// TwinCAT 3 PLC project MU
// ProgramVersion: 3.1.4026.14
// libraries:
//   Tc2_ControllerToolbox, * (Beckhoff Automation GmbH)
//   Tc2_ModbusRTU, * (Beckhoff Automation GmbH)
//   Tc2_SerialCom, * (Beckhoff Automation GmbH)
//   Tc2_Standard, * (Beckhoff Automation GmbH)
//   Tc2_System, * (Beckhoff Automation GmbH)
//   Tc2_Utilities, * (Beckhoff Automation GmbH)
//   Tc3_Module, * (Beckhoff Automation GmbH)
// project tree:
//   DATA TYPES/ E_ComState.TcDUT, E_MFC_INDEX.TcDUT, E_MFC_MESSAGE.TcDUT (not stored), ST_MfcData.TcDUT (not stored)
//   DATA TYPES/MODUELS/ ST_GAS_CABINET.TcDUT (not stored), ST_MAIN_MODULE.TcDUT, ST_NOTIFICATION.TcDUT, ST_NOTIFICATION_MESSAGE.TcDUT (not stored), ST_REACTOR_CABINET.TcDUT, ST_SEQUENCE.TcDUT, ST_SOL_VALVE.TcDUT (not stored), ST_TEMP_CONTROLLER.TcDUT, ST_THROTTLE_VALVE.TcDUT, ST_UTILITY.TcDUT, ST_ROTATION_MOTOR.TcDUT
//   DATA TYPES/PARTS/ ST_ANALOG_PART.TcDUT, ST_DIGITAL_PART.TcDUT, ST_SEQUENCE_PART.TcDUT
//   DEVICE/LINE HEATER/ FB_LINE_HEATER_MANAGER.TcPOU (not stored), FB_Modbus_Send_FIFO.TcPOU (not stored), FB_TEMP_RAMPING.TcPOU
//   DEVICE/LINE HEATER/FUNCTION/ F_Temp_Write_Set_Point.TcPOU (not stored), F_Temp_Write_Value.TcPOU
//   DEVICE/ ST_LineHeater_Data.TcDUT, ST_Modbus_Send_Frame.TcDUT
//   DUTs/ AnalogController.TcDUT, E_ControlMode.TcDUT (not stored), E_RampGeneratorState.TcDUT (not stored), E_RecipeRun.TcDUT (not stored), E_RecipeRunETMode.TcDUT (not stored), E_TowerLamp.TcDUT (not stored), GeneralIO.TcDUT, MainPRGControl.TcDUT, OperationMode.TcDUT (not stored), outWord.TcDUT (not stored), RampGeneratorInput.TcDUT (not stored)
//   DUTs/DUTs/ENUM/ E_aAnalogInputIO_Index.TcDUT, E_AlarmList.TcDUT, E_AlarmSetValue.TcDUT (not stored), E_InputState.TcDUT, E_Interlock.TcDUT, E_Morning_Index.TcDUT, E_WarningList.TcDUT (not stored)
//   DUTs/DUTs/ F_GetReal_USINT.TcDUT
//   DUTs/Interlock/ Interlock.TcDUT, InterlockEnableThreshold.TcDUT, InterlockSetting.TcDUT, InterlockState.TcDUT, LogicalInterlockSubstate.TcDUT
//   DUTs/IO/ AnalogIO.TcDUT, DigitalIO.TcDUT, IO.TcDUT
//   DUTs/Recipe/ Recipe.TcDUT, RecipeControl.TcDUT, RecipeRunET.TcDUT (not stored), RecipeStep.TcDUT, ScaleFactor.TcDUT
//   FUNCTION/ BOOL_TO_STRING_LHeaterON.TcPOU, CheckRangeSigned.TcPOU (not stored), CheckRangeUnsigned.TcPOU (not stored), FB_TON_Pausable.TcPOU (not stored), F_GetDorPressure.TcPOU, F_State_All_Valve_Vent.TcPOU (not stored), HEXSTR_TO_REAL_LHeaterPV.TcPOU (not stored), F_ReactorIndexToAnalogControllerIndex.TcPOU, Real_To_String_LineHeater.TcPOU, Real_To_String_ThermalBath.TcPOU (not stored), USINT_TO_WORD_Bit.TcPOU (not stored), USINT_TO_WORD_jh.TcPOU, WORD_TO_USINT_Bit.TcPOU (not stored)
//   GVLs/ GVL_INTERFACE_UI.TcGVL, GVL_COMMAND_FROM_UI.TcGVL (not stored), GVL_CONSTANT.TcGVL, GVL_DEVICE_NET_E3508.TcGVL, GVL_DEVICE_NET_IQ_PLUS.TcGVL, GVL_IO.TcGVL, GVL.TcGVL, GVL_IO_GAS_CABINET.TcGVL, GVL_IO_REACTOR_CABINET.TcGVL, GVL_IO_VALVE.TcGVL (not stored), GVL_PERSISTENT.TcGVL (not stored), GVL_SEQUENCE.TcGVL (not stored), GVL_Serial.TcGVL
//   / PlcTask.TcTTO (not stored)
//   POUs/ FB_AnalogDeviceRampControl.TcPOU, FB_ControlRampGenerator.TcPOU (not stored), FB_DeviationCheck.TcPOU (not stored), FB_FaultCheck.TcPOU (not stored), FB_OverLimitCheck.TcPOU, FB_RecipeAnalogControlInputSequencer.TcPOU, F_StopAnalogRamping_ForRecipe.TcPOU, FB_SensorLimitCheck.TcPOU (not stored), FB_ValveControl.TcPOU, F_ResetTimersAndRCPTimes.TcPOU (not stored), MAIN.TcPOU, P11_E3508.TcPOU, P12_IQ_PLUS.TcPOU, P13_LineHeater.TcPOU, P14_ThermalBath.TcPOU, P15_RotationOperation.TcPOU, P16_CoverOperation.TcPOU, P17_DOROperation.TcPOU, P22_Background_ThermalBath.TcPOU, P30_ManualControl.TcPOU (not stored), P31_PriorityControl.TcPOU, P50_RecipeControl.TcPOU, P60_UpdatePV.TcPOU, P70_Interface.TcPOU (not stored), P90_Interlock.TcPOU, P91_Monitoring.TcPOU, P92_Maintenance.TcPOU
//   POUs/FUNCTION/ FB_RINGBUFFER.TcPOU, F_StateValve_Process_Source.TcPOU, F_StateValve_Process.TcPOU
//   POUs/VARIABLE_LINK/ F_Variable_DeviceLink.TcPOU, F_Variable_Valve.TcPOU, F_Variable_FromUI.TcPOU, F_Variable_FromUI_Interlock.TcPOU, F_Variable_TODevice.TcPOU (not stored), F_Variable_ToUI_InputState.TcPOU
// real-time tasks:
//   TASK PlcTask: cycle T#10ms, priority 20, ADS port 350
// I/O:
//   DEVICE Device 1 (EtherCAT) (disabled), AmsNetId 192.168.123.106.2.1
//     Term 1 (EK1200) [EK1200-5000 EtherCAT Power supply (2A E-Bus)]
//       Term 2 (EL1088) [EL1088 8Ch. Dig. Input 24V, 3ms, negative]
//       Term 3 (EL1088) [EL1088 8Ch. Dig. Input 24V, 3ms, negative]
//       Term 4 (EL1088) [EL1088 8Ch. Dig. Input 24V, 3ms, negative]
//       Term 5 (EL1088) [EL1088 8Ch. Dig. Input 24V, 3ms, negative]
//       Term 6 (EL1088) [EL1088 8Ch. Dig. Input 24V, 3ms, negative]
//       Term 7 (EL1088) [EL1088 8Ch. Dig. Input 24V, 3ms, negative]
//       Term 8 (EL2088) [EL2088 8Ch. Dig. Output 24V, 0.5A, switching to negative]
//       Term 9 (EL2088) [EL2088 8Ch. Dig. Output 24V, 0.5A, switching to negative]
//       Term 10 (EL3064) [EL3064 4Ch. Ana. Input 0-10V]
//       Term 11 (EL4004) [EL4004 4Ch. Ana. Output 0-10V, 12bit]
//       Term 12 (EL9410) [EL9410 E-Bus Power Supplier  (Diagnostics)]
//       Term 13 (EL3064) [EL3064 4Ch. Ana. Input 0-10V]
//       Term 14 (EL4004) [EL4004 4Ch. Ana. Output 0-10V, 12bit]
//       Term 15 (EL3064) [EL3064 4Ch. Ana. Input 0-10V]
//       Term 16 (EL4004) [EL4004 4Ch. Ana. Output 0-10V, 12bit]
//       Term 17 (EL3064) [EL3064 4Ch. Ana. Input 0-10V]
//       Term 18 (EL4004) [EL4004 4Ch. Ana. Output 0-10V, 12bit]
//       Term 19 (EL3102) [EL3102 2Ch. Ana. Input +/-10V, Diff.]
//       Term 20 (EL3024) [EL3024 4Ch. Ana. Input 4-20mA DIFF]
//       Term 21 (EL6021) [EL6021 Interface (RS422/485)]
//       Term 22 (EL6021) [EL6021 Interface (RS422/485)]
//       Term 23 (EL6752) [EL6752 DeviceNet Master]
//       Term 24 (EK1110) [EK1110 EtherCAT extension]
//     Term 25 (EK1100) [EK1100 EtherCAT Coupler (2A E-Bus)]
//       Term 26 (EL1088) [EL1088 8Ch. Dig. Input 24V, 3ms, negative]
//       Term 27 (EL1088) [EL1088 8Ch. Dig. Input 24V, 3ms, negative]
//       Term 28 (EL1088) [EL1088 8Ch. Dig. Input 24V, 3ms, negative]
//       Term 29 (EL2088) [EL2088 8Ch. Dig. Output 24V, 0.5A, switching to negative]
//       Term 30 (EL2088) [EL2088 8Ch. Dig. Output 24V, 0.5A, switching to negative]
//       Term 31 (EL2088) [EL2088 8Ch. Dig. Output 24V, 0.5A, switching to negative]
//       Term 32 (EL3064) [EL3064 4Ch. Ana. Input 0-10V]
//       Term 33 (EL3024) [EL3024 4Ch. Ana. Input 4-20mA DIFF]
//       Term 34 (EL4004) [EL4004 4Ch. Ana. Output 0-10V, 12bit]
//       Term 35 (EL3204) [EL3204 4Ch. Ana. Input PT100 (RTD)]
//       Term 36 (EL9011) [EL9011 End Terminal]
//   DEVICE Device 2 (EL6752) (disabled), AmsNetId 192.168.123.106.3.1
//     SolValve // EDS-File: 'OPP6-2D.EDS' DescText: OPP6-2D Vendor: CKD Corporation Device Type: Generic Device Product Name: OPP6-2D Catalog Number:
//     ThrottleValve // EDS-File: 'TBJQPDNG-L041X01 155OUT154.EDS' DescText: Intellisys IQ-Plus Vendor: Nor-Cal Products Device Type: Process Control Valve Product Name: INTELLISYS Catalog Number: IQ-Plus
//     TempController // EDS-File: '3500-2.3V2.EDS' DescText: Eurotherm 3500 Vendor: Eurotherm Device Type: Generic Product Name: Eurotherm 3500 Catalog Number:
// variable links:
//   MU/MU Instance <-> Device 1 (EtherCAT)/Term 1 (EK1200)/Term 10 (EL3064)
//     PlcTask Inputs/GVL_IO_GAS_CABINET.AI_09_M01_ChalcogenRunPV <-> AI Standard Channel 1/Value
//     PlcTask Inputs/GVL_IO_GAS_CABINET.AI_09_M02_MORunPV <-> AI Standard Channel 2/Value
//     PlcTask Inputs/GVL_IO_GAS_CABINET.AI_09_M03_H2SeSupplyPV <-> AI Standard Channel 3/Value
//     PlcTask Inputs/GVL_IO_GAS_CABINET.AI_09_M04_H2SSupplyPV <-> AI Standard Channel 4/Value
//   MU/MU Instance <-> Device 1 (EtherCAT)/Term 1 (EK1200)/Term 11 (EL4004)
//     PlcTask Outputs/GVL_IO_GAS_CABINET.AO_10_M01_ChalcogenRunSV <-> AO Outputs Channel 1/Analog output
//     PlcTask Outputs/GVL_IO_GAS_CABINET.AO_10_M02_MORunSV <-> AO Outputs Channel 2/Analog output
//     PlcTask Outputs/GVL_IO_GAS_CABINET.AO_10_M03_H2SeSupplySV <-> AO Outputs Channel 3/Analog output
//     PlcTask Outputs/GVL_IO_GAS_CABINET.AO_10_M04_H2SSupplySV <-> AO Outputs Channel 4/Analog output
//   MU/MU Instance <-> Device 1 (EtherCAT)/Term 1 (EK1200)/Term 13 (EL3064)
//     PlcTask Inputs/GVL_IO_GAS_CABINET.AI_11_M05_Source_1TMInSupplyPV <-> AI Standard Channel 1/Value
//     PlcTask Inputs/GVL_IO_GAS_CABINET.AI_11_M06_Source_2TMGaSupplyPV <-> AI Standard Channel 2/Value
//     PlcTask Inputs/GVL_IO_GAS_CABINET.AI_11_M07_Source_3DMSeSupplyPV <-> AI Standard Channel 3/Value
//     PlcTask Inputs/GVL_IO_GAS_CABINET.AI_11_M08_Source_4ChalcoSupplyPV <-> AI Standard Channel 4/Value
//   MU/MU Instance <-> Device 1 (EtherCAT)/Term 1 (EK1200)/Term 14 (EL4004)
//     PlcTask Outputs/GVL_IO_GAS_CABINET.AO_12_M05_Source_1TMInSupplySV <-> AO Outputs Channel 1/Analog output
//     PlcTask Outputs/GVL_IO_GAS_CABINET.AO_12_M06_Source_2TMGaSupplySV <-> AO Outputs Channel 2/Analog output
//     PlcTask Outputs/GVL_IO_GAS_CABINET.AO_12_M07_Source_3DMSeSupplySV <-> AO Outputs Channel 3/Analog output
//     PlcTask Outputs/GVL_IO_GAS_CABINET.AO_12_M08_Source_4ChalcoSupplySV <-> AO Outputs Channel 4/Analog output
//   MU/MU Instance <-> Device 1 (EtherCAT)/Term 1 (EK1200)/Term 15 (EL3064)
//     PlcTask Inputs/GVL_IO_GAS_CABINET.AI_13_M09_LinerPurgePV <-> AI Standard Channel 1/Value
//     PlcTask Inputs/GVL_IO_GAS_CABINET.AI_13_M10_HeaterPurgePV <-> AI Standard Channel 2/Value
//     PlcTask Inputs/GVL_IO_GAS_CABINET.AI_13_M11_ChalcogenVentPV <-> AI Standard Channel 3/Value
//     PlcTask Inputs/GVL_IO_GAS_CABINET.AI_13_M12_MOVentPV <-> AI Standard Channel 4/Value
//   MU/MU Instance <-> Device 1 (EtherCAT)/Term 1 (EK1200)/Term 16 (EL4004)
//     PlcTask Outputs/GVL_IO_GAS_CABINET.AO_14_M09_LinerPurgeSV <-> AO Outputs Channel 1/Analog output
//     PlcTask Outputs/GVL_IO_GAS_CABINET.AO_14_M10_HeaterPurgeSV <-> AO Outputs Channel 2/Analog output
//     PlcTask Outputs/GVL_IO_GAS_CABINET.AO_14_M11_ChalcogenVentSV <-> AO Outputs Channel 3/Analog output
//     PlcTask Outputs/GVL_IO_GAS_CABINET.AO_14_M12_MOVentSV <-> AO Outputs Channel 4/Analog output
//   MU/MU Instance <-> Device 1 (EtherCAT)/Term 1 (EK1200)/Term 17 (EL3064)
//     PlcTask Inputs/GVL_IO_GAS_CABINET.AI_15_E01Source_1TMInPressurePV <-> AI Standard Channel 1/Value
//     PlcTask Inputs/GVL_IO_GAS_CABINET.AI_15_E02Source_2TMGaPressurePV <-> AI Standard Channel 2/Value
//     PlcTask Inputs/GVL_IO_GAS_CABINET.AI_15_E03Source_3DMSePressurePV <-> AI Standard Channel 3/Value
//     PlcTask Inputs/GVL_IO_GAS_CABINET.AI_15_E04Source_4ChalcoPressurePV <-> AI Standard Channel 4/Value
//   MU/MU Instance <-> Device 1 (EtherCAT)/Term 1 (EK1200)/Term 18 (EL4004)
//     PlcTask Outputs/GVL_IO_GAS_CABINET.AO_16_E01Source_1TMInPressureSV <-> AO Outputs Channel 1/Analog output
//     PlcTask Outputs/GVL_IO_GAS_CABINET.AO_16_E02Source_2TMGaPressureSV <-> AO Outputs Channel 2/Analog output
//     PlcTask Outputs/GVL_IO_GAS_CABINET.AO_16_E03Source_3DMSePressureSV <-> AO Outputs Channel 3/Analog output
//     PlcTask Outputs/GVL_IO_GAS_CABINET.AO_16_E04Source_4ChalcoPressureSV <-> AO Outputs Channel 4/Analog output
//   MU/MU Instance <-> Device 1 (EtherCAT)/Term 1 (EK1200)/Term 19 (EL3102)
//     PlcTask Inputs/GVL_IO_GAS_CABINET.DI_17_DP1ChalcogenDP <-> AI Standard Channel 1/Value
//     PlcTask Inputs/GVL_IO_GAS_CABINET.DI_17_DP2MODP <-> AI Standard Channel 2/Value
//   MU/MU Instance <-> Device 1 (EtherCAT)/Term 1 (EK1200)/Term 2 (EL1088)
//     PlcTask Inputs/GVL_IO_GAS_CABINET.DI_01_ControlCabinetDoorClose <-> Channel 5/Input
//     PlcTask Inputs/GVL_IO_GAS_CABINET.DI_01_GasCabinetDoorClose <-> Channel 4/Input
//     PlcTask Inputs/GVL_IO_GAS_CABINET.DI_01_GasCabinetLampButton <-> Channel 2/Input
//     PlcTask Inputs/GVL_IO_GAS_CABINET.DI_01_PneumaticPressureSensor <-> Channel 3/Input
//     PlcTask Inputs/GVL_IO_GAS_CABINET.DI_01_ResetButton <-> Channel 1/Input
//     PlcTask Inputs/GVL_IO_GAS_CABINET.DI_01_SMPS_1Alarm <-> Channel 6/Input
//     PlcTask Inputs/GVL_IO_GAS_CABINET.DI_01_SMPS_2Alarm <-> Channel 7/Input
//     PlcTask Inputs/GVL_IO_GAS_CABINET.DI_01_SMPS_3Alarm <-> Channel 8/Input
//   MU/MU Instance <-> Device 1 (EtherCAT)/Term 1 (EK1200)/Term 20 (EL3024)
//     PlcTask Inputs/GVL_IO_GAS_CABINET.DI_18_S01N2SupplyPressPV <-> AI Standard Channel 1/Value
//     PlcTask Inputs/GVL_IO_GAS_CABINET.DI_18_S02H2SupplyPressPV <-> AI Standard Channel 2/Value
//     PlcTask Inputs/GVL_IO_GAS_CABINET.DI_18_S03H2SSupplyPressPV <-> AI Standard Channel 3/Value
//     PlcTask Inputs/GVL_IO_GAS_CABINET.DI_18_S04H2SeSupplyPressPV <-> AI Standard Channel 4/Value
//   MU/MU Instance <-> Device 1 (EtherCAT)/Term 1 (EK1200)/Term 21 (EL6021)
//     PlcTask Inputs/GVL.fbLineHeater_Manager.fbModbus_Master.InData/D <-> COM TxPDO-Map Inputs/Data In 0
//     PlcTask Inputs/GVL.fbLineHeater_Manager.fbModbus_Master.InData/D @bit {8..168 step 8} <-> COM TxPDO-Map Inputs/Data In {1..21}  (21 links)
//     PlcTask Inputs/GVL.fbLineHeater_Manager.fbModbus_Master.InData/Status <-> COM TxPDO-Map Inputs/Status
//     PlcTask Outputs/GVL.fbLineHeater_Manager.fbModbus_Master.OutData/Ctrl <-> COM RxPDO-Map Outputs/Ctrl
//     PlcTask Outputs/GVL.fbLineHeater_Manager.fbModbus_Master.OutData/D <-> COM RxPDO-Map Outputs/Data Out 0
//     PlcTask Outputs/GVL.fbLineHeater_Manager.fbModbus_Master.OutData/D @bit {8..168 step 8} <-> COM RxPDO-Map Outputs/Data Out {1..21}  (21 links)
//   MU/MU Instance <-> Device 1 (EtherCAT)/Term 1 (EK1200)/Term 22 (EL6021)
//     PlcTask Inputs/GVL_Serial.stIn_KL6031_TB/D <-> COM TxPDO-Map Inputs/Data In 0
//     PlcTask Inputs/GVL_Serial.stIn_KL6031_TB/D @bit {8..168 step 8} <-> COM TxPDO-Map Inputs/Data In {1..21}  (21 links)
//     PlcTask Inputs/GVL_Serial.stIn_KL6031_TB/Status <-> COM TxPDO-Map Inputs/Status
//     PlcTask Outputs/GVL_Serial.stOut_KL6031_TB/Ctrl <-> COM RxPDO-Map Outputs/Ctrl
//     PlcTask Outputs/GVL_Serial.stOut_KL6031_TB/D <-> COM RxPDO-Map Outputs/Data Out 0
//     PlcTask Outputs/GVL_Serial.stOut_KL6031_TB/D @bit {8..168 step 8} <-> COM RxPDO-Map Outputs/Data Out {1..21}  (21 links)
//   MU/MU Instance <-> Device 1 (EtherCAT)/Term 1 (EK1200)/Term 3 (EL1088)
//     PlcTask Inputs/GVL_IO_GAS_CABINET.DI_02_CoverLiftMotorCP <-> Channel 7/Input
//     PlcTask Inputs/GVL_IO_GAS_CABINET.DI_02_GraphiteHeaterELCB <-> Channel 2/Input
//     PlcTask Inputs/GVL_IO_GAS_CABINET.DI_02_LineHeatersELCB <-> Channel 5/Input
//     PlcTask Inputs/GVL_IO_GAS_CABINET.DI_02_RotationMotorCP <-> Channel 6/Input
//     PlcTask Inputs/GVL_IO_GAS_CABINET.DI_02_SMPS_4Alarm <-> Channel 1/Input
//     PlcTask Inputs/GVL_IO_GAS_CABINET.DI_02_T_VCP <-> Channel 8/Input
//     PlcTask Inputs/GVL_IO_GAS_CABINET.DI_02_ThermalBathsELCB <-> Channel 3/Input
//     PlcTask Inputs/GVL_IO_GAS_CABINET.DI_02_VacuumPumpELCB <-> Channel 4/Input
//   MU/MU Instance <-> Device 1 (EtherCAT)/Term 1 (EK1200)/Term 4 (EL1088)
//     PlcTask Inputs/GVL_IO_GAS_CABINET.DI_03_CabinetLampsCP <-> Channel 2/Input
//     PlcTask Inputs/GVL_IO_GAS_CABINET.DI_03_GasDetectorCP <-> Channel 1/Input
//     PlcTask Inputs/GVL_IO_GAS_CABINET.DI_03_LineHeater_1CP <-> Channel 4/Input
//     PlcTask Inputs/GVL_IO_GAS_CABINET.DI_03_LineHeater_2CP <-> Channel 5/Input
//     PlcTask Inputs/GVL_IO_GAS_CABINET.DI_03_LineHeater_3CP <-> Channel 6/Input
//     PlcTask Inputs/GVL_IO_GAS_CABINET.DI_03_LineHeater_4CP <-> Channel 7/Input
//     PlcTask Inputs/GVL_IO_GAS_CABINET.DI_03_LineHeater_5CP <-> Channel 8/Input
//     PlcTask Inputs/GVL_IO_GAS_CABINET.DI_03_MFCPowerCP <-> Channel 3/Input
//   MU/MU Instance <-> Device 1 (EtherCAT)/Term 1 (EK1200)/Term 5 (EL1088)
//     PlcTask Inputs/GVL_IO_GAS_CABINET.DI_04_ExternalScrubberFault <-> Channel 8/Input
//     PlcTask Inputs/GVL_IO_GAS_CABINET.DI_04_FireSensor <-> Channel 7/Input
//     PlcTask Inputs/GVL_IO_GAS_CABINET.DI_04_GasDetectorH2 <-> Channel 4/Input
//     PlcTask Inputs/GVL_IO_GAS_CABINET.DI_04_GasDetectorH2S <-> Channel 5/Input
//     PlcTask Inputs/GVL_IO_GAS_CABINET.DI_04_GasDetectorH2Se <-> Channel 6/Input
//     PlcTask Inputs/GVL_IO_GAS_CABINET.DI_04_LineHeater_6CP <-> Channel 1/Input
//     PlcTask Inputs/GVL_IO_GAS_CABINET.DI_04_LineHeater_7CP <-> Channel 2/Input
//     PlcTask Inputs/GVL_IO_GAS_CABINET.DI_04_LineHeater_8CP <-> Channel 3/Input
//   MU/MU Instance <-> Device 1 (EtherCAT)/Term 1 (EK1200)/Term 6 (EL1088)
//     PlcTask Inputs/GVL_IO_GAS_CABINET.DI_05_ExternalH2GasCabinetFault <-> Channel 1/Input
//     PlcTask Inputs/GVL_IO_GAS_CABINET.DI_05_ExternalH2SGasCabinetFault <-> Channel 2/Input
//     PlcTask Inputs/GVL_IO_GAS_CABINET.DI_05_ExternalH2SeGasCabinetFault <-> Channel 3/Input
//     PlcTask Inputs/GVL_IO_GAS_CABINET.DI_05_ExternalUserInputAlarm <-> Channel 4/Input
//     PlcTask Inputs/GVL_IO_GAS_CABINET.DI_05_ThermalBath_1CutOffAlarm <-> Channel 6/Input
//     PlcTask Inputs/GVL_IO_GAS_CABINET.DI_05_ThermalBath_2CutOffAlarm <-> Channel 8/Input
//     PlcTask Inputs/GVL_IO_GAS_CABINET.DI_05_ThermalBath_1DeviationAlarm <-> Channel 5/Input
//     PlcTask Inputs/GVL_IO_GAS_CABINET.DI_05_ThermalBath_2DeviationAlarm <-> Channel 7/Input
//   MU/MU Instance <-> Device 1 (EtherCAT)/Term 1 (EK1200)/Term 7 (EL1088)
//     PlcTask Inputs/GVL_IO_GAS_CABINET.DI_06_Spare_01 <-> Channel 5/Input
//     PlcTask Inputs/GVL_IO_GAS_CABINET.DI_06_Spare_02 <-> Channel 6/Input
//     PlcTask Inputs/GVL_IO_GAS_CABINET.DI_06_Spare_03 <-> Channel 7/Input
//     PlcTask Inputs/GVL_IO_GAS_CABINET.DI_06_Spare_04 <-> Channel 8/Input
//     PlcTask Inputs/GVL_IO_GAS_CABINET.DI_06_ThermalBath_3CutOffAlarm <-> Channel 2/Input
//     PlcTask Inputs/GVL_IO_GAS_CABINET.DI_06_ThermalBath_4CutOffAlarm <-> Channel 4/Input
//     PlcTask Inputs/GVL_IO_GAS_CABINET.DI_06_ThermalBath_3DeviationAlarm <-> Channel 1/Input
//     PlcTask Inputs/GVL_IO_GAS_CABINET.DI_06_ThermalBath_4DeviationAlarm <-> Channel 3/Input
//   MU/MU Instance <-> Device 1 (EtherCAT)/Term 1 (EK1200)/Term 8 (EL2088)
//     PlcTask Outputs/GVL_IO_GAS_CABINET.DO_07_ControlCabinetLamp <-> Channel 2/Output
//     PlcTask Outputs/GVL_IO_GAS_CABINET.DO_07_GasCabinetLamp <-> Channel 3/Output
//     PlcTask Outputs/GVL_IO_GAS_CABINET.DO_07_GraphiteHeaterMC <-> Channel 4/Output
//     PlcTask Outputs/GVL_IO_GAS_CABINET.DO_07_LineHeatersMC <-> Channel 7/Output
//     PlcTask Outputs/GVL_IO_GAS_CABINET.DO_07_ResetButtonLamp <-> Channel 8/Output
//     PlcTask Outputs/GVL_IO_GAS_CABINET.DO_07_SystemPowerOffLock <-> Channel 1/Output
//     PlcTask Outputs/GVL_IO_GAS_CABINET.DO_07_ThermalBathsMC <-> Channel 5/Output
//     PlcTask Outputs/GVL_IO_GAS_CABINET.DO_07_VacuumPumpMC <-> Channel 6/Output
//   MU/MU Instance <-> Device 1 (EtherCAT)/Term 1 (EK1200)/Term 9 (EL2088)
//     PlcTask Outputs/GVL_IO_GAS_CABINET.DO_08_Spare_01 <-> Channel 1/Output
//     PlcTask Outputs/GVL_IO_GAS_CABINET.DO_08_Spare_02 <-> Channel 2/Output
//     PlcTask Outputs/GVL_IO_GAS_CABINET.DO_08_Spare_03 <-> Channel 3/Output
//     PlcTask Outputs/GVL_IO_GAS_CABINET.DO_08_Spare_04 <-> Channel 4/Output
//     PlcTask Outputs/GVL_IO_GAS_CABINET.DO_08_Spare_05 <-> Channel 5/Output
//     PlcTask Outputs/GVL_IO_GAS_CABINET.DO_08_Spare_06 <-> Channel 6/Output
//     PlcTask Outputs/GVL_IO_GAS_CABINET.DO_08_Spare_07 <-> Channel 7/Output
//     PlcTask Outputs/GVL_IO_GAS_CABINET.DO_08_Spare_08 <-> Channel 8/Output
//   MU/MU Instance <-> Device 1 (EtherCAT)/Term 25 (EK1100)/Term 26 (EL1088)
//     PlcTask Inputs/GVL_IO_REACTOR_CABINET.DI_01_ClampLock <-> Channel 7/Input
//     PlcTask Inputs/GVL_IO_REACTOR_CABINET.DI_01_ClampRelease <-> Channel 8/Input
//     PlcTask Inputs/GVL_IO_REACTOR_CABINET.DI_01_DORATMButton <-> Channel 4/Input
//     PlcTask Inputs/GVL_IO_REACTOR_CABINET.DI_01_DORVACButton <-> Channel 3/Input
//     PlcTask Inputs/GVL_IO_REACTOR_CABINET.DI_01_MaintenanceModeKey <-> Channel 1/Input
//     PlcTask Inputs/GVL_IO_REACTOR_CABINET.DI_01_ReactorCabinetLampButton <-> Channel 2/Input
//     PlcTask Inputs/GVL_IO_REACTOR_CABINET.DI_01_ReactorDoorDownButton <-> Channel 6/Input
//     PlcTask Inputs/GVL_IO_REACTOR_CABINET.DI_01_ReactorDoorUpButton <-> Channel 5/Input
//   MU/MU Instance <-> Device 1 (EtherCAT)/Term 25 (EK1100)/Term 27 (EL1088)
//     PlcTask Inputs/GVL_IO_REACTOR_CABINET.DI_02_C_WFlowSensor <-> Channel 1/Input
//     PlcTask Inputs/GVL_IO_REACTOR_CABINET.DI_02_ReactorDoorUpLimitSensor <-> Channel 8/Input
//     PlcTask Inputs/GVL_IO_REACTOR_CABINET.DI_02_SusceptorRotationMotorFault <-> Channel 2/Input
//     PlcTask Inputs/GVL_IO_REACTOR_CABINET.DI_02_VacuumPumpAlarm <-> Channel 5/Input
//     PlcTask Inputs/GVL_IO_REACTOR_CABINET.DI_02_VacuumPumpFBRunning <-> Channel 7/Input
//     PlcTask Inputs/GVL_IO_REACTOR_CABINET.DI_02_VacuumPumpFail <-> Channel 3/Input
//     PlcTask Inputs/GVL_IO_REACTOR_CABINET.DI_02_VacuumPumpRunning <-> Channel 6/Input
//     PlcTask Inputs/GVL_IO_REACTOR_CABINET.DI_02_VacuumPumpWarning <-> Channel 4/Input
//   MU/MU Instance <-> Device 1 (EtherCAT)/Term 25 (EK1100)/Term 28 (EL1088)
//     PlcTask Inputs/GVL_IO_REACTOR_CABINET.DI_03_CylinderAutoSwitch_Closed <-> Channel 2/Input
//     PlcTask Inputs/GVL_IO_REACTOR_CABINET.DI_03_CylinderAutoSwitch_Opened <-> Channel 3/Input
//     PlcTask Inputs/GVL_IO_REACTOR_CABINET.DI_03_ReactorCabinetDoorClose <-> Channel 4/Input
//     PlcTask Inputs/GVL_IO_REACTOR_CABINET.DI_03_ReactorDoorDownLimitSensor <-> Channel 1/Input
//     PlcTask Inputs/GVL_IO_REACTOR_CABINET.DI_03_Spare_01 <-> Channel 5/Input
//     PlcTask Inputs/GVL_IO_REACTOR_CABINET.DI_03_Spare_02 <-> Channel 6/Input
//     PlcTask Inputs/GVL_IO_REACTOR_CABINET.DI_03_Spare_03 <-> Channel 7/Input
//     PlcTask Inputs/GVL_IO_REACTOR_CABINET.DI_03_Spare_04 <-> Channel 8/Input
//   MU/MU Instance <-> Device 1 (EtherCAT)/Term 25 (EK1100)/Term 29 (EL2088)
//     PlcTask Outputs/GVL_IO_REACTOR_CABINET.DO_04_ReactorCoverDownRelay <-> Channel 8/Output
//     PlcTask Outputs/GVL_IO_REACTOR_CABINET.DO_04_ReactorCoverUpRelay <-> Channel 7/Output
//     PlcTask Outputs/GVL_IO_REACTOR_CABINET.DO_04_SignalTowerBlue <-> Channel 4/Output
//     PlcTask Outputs/GVL_IO_REACTOR_CABINET.DO_04_SignalTowerBuzzer <-> Channel 6/Output
//     PlcTask Outputs/GVL_IO_REACTOR_CABINET.DO_04_SignalTowerGreen <-> Channel 3/Output
//     PlcTask Outputs/GVL_IO_REACTOR_CABINET.DO_04_SignalTowerOrange <-> Channel 2/Output
//     PlcTask Outputs/GVL_IO_REACTOR_CABINET.DO_04_SignalTowerRed <-> Channel 1/Output
//     PlcTask Outputs/GVL_IO_REACTOR_CABINET.DO_04_SignalTowerWhite <-> Channel 5/Output
//   MU/MU Instance <-> Device 1 (EtherCAT)/Term 25 (EK1100)/Term 30 (EL2088)
//     PlcTask Outputs/GVL_IO_REACTOR_CABINET.DO_05_ClampLock <-> Channel 1/Output
//     PlcTask Outputs/GVL_IO_REACTOR_CABINET.DO_05_ClampRelease <-> Channel 2/Output
//     PlcTask Outputs/GVL_IO_REACTOR_CABINET.DO_05_DORVACButtonLamp <-> Channel 8/Output
//     PlcTask Outputs/GVL_IO_REACTOR_CABINET.DO_05_SusceptorRotationAL_RST <-> Channel 7/Output
//     PlcTask Outputs/GVL_IO_REACTOR_CABINET.DO_05_SusceptorRotationFWD <-> Channel 5/Output
//     PlcTask Outputs/GVL_IO_REACTOR_CABINET.DO_05_SusceptorRotationSTOP <-> Channel 6/Output
//     PlcTask Outputs/GVL_IO_REACTOR_CABINET.DO_05_VacuumPumpReset <-> Channel 4/Output
//     PlcTask Outputs/GVL_IO_REACTOR_CABINET.DO_05_VacuumPumpStart_Stop <-> Channel 3/Output
//   MU/MU Instance <-> Device 1 (EtherCAT)/Term 25 (EK1100)/Term 31 (EL2088)
//     PlcTask Outputs/GVL_IO_REACTOR_CABINET.DO_06_ClampLockButtonLamp <-> Channel 4/Output
//     PlcTask Outputs/GVL_IO_REACTOR_CABINET.DO_06_ClampReleaseButtonLamp <-> Channel 5/Output
//     PlcTask Outputs/GVL_IO_REACTOR_CABINET.DO_06_DORATMButtonLamp <-> Channel 1/Output
//     PlcTask Outputs/GVL_IO_REACTOR_CABINET.DO_06_ReactorCabinetLamp <-> Channel 6/Output
//     PlcTask Outputs/GVL_IO_REACTOR_CABINET.DO_06_ReactorCoverDownButtonLamp <-> Channel 3/Output
//     PlcTask Outputs/GVL_IO_REACTOR_CABINET.DO_06_ReactorCoverUpButtonLamp <-> Channel 2/Output
//     PlcTask Outputs/GVL_IO_REACTOR_CABINET.DO_06_Spare07 <-> Channel 7/Output
//     PlcTask Outputs/GVL_IO_REACTOR_CABINET.DO_06_Spare08 <-> Channel 8/Output
//   MU/MU Instance <-> Device 1 (EtherCAT)/Term 25 (EK1100)/Term 32 (EL3064)
//     PlcTask Inputs/GVL_IO_REACTOR_CABINET.AI_07_P02_ReactorPressure10TorrPV <-> AI Standard Channel 1/Value
//     PlcTask Inputs/GVL_IO_REACTOR_CABINET.AI_07_P03_ExhaustPressurePV <-> AI Standard Channel 3/Value
//     PlcTask Inputs/GVL_IO_REACTOR_CABINET.AI_07_S05_DORPressurePV <-> AI Standard Channel 2/Value
//     PlcTask Inputs/GVL_IO_REACTOR_CABINET.AI_07_Spare_04 <-> AI Standard Channel 4/Value
//   MU/MU Instance <-> Device 1 (EtherCAT)/Term 25 (EK1100)/Term 33 (EL3024)
//     PlcTask Inputs/GVL_IO_REACTOR_CABINET.AI_08_R01SusceptorRotationPV <-> AI Standard Channel 1/Value
//     PlcTask Inputs/GVL_IO_REACTOR_CABINET.AI_08_Spare_02 <-> AI Standard Channel 2/Value
//     PlcTask Inputs/GVL_IO_REACTOR_CABINET.AI_08_Spare_03 <-> AI Standard Channel 3/Value
//     PlcTask Inputs/GVL_IO_REACTOR_CABINET.AI_08_Spare_04 <-> AI Standard Channel 4/Value
//   MU/MU Instance <-> Device 1 (EtherCAT)/Term 25 (EK1100)/Term 34 (EL4004)
//     PlcTask Outputs/GVL_IO_REACTOR_CABINET.AO_09_P03_ExhaustPressureAM215Input <-> AO Outputs Channel 1/Analog output
//     PlcTask Outputs/GVL_IO_REACTOR_CABINET.AO_09_R01_SusceptorRotationSV <-> AO Outputs Channel 2/Analog output
//     PlcTask Outputs/GVL_IO_REACTOR_CABINET.AO_09_Spare_03 <-> AO Outputs Channel 3/Analog output
//     PlcTask Outputs/GVL_IO_REACTOR_CABINET.AO_09_Spare_04 <-> AO Outputs Channel 4/Analog output
//   MU/MU Instance <-> Device 1 (EtherCAT)/Term 25 (EK1100)/Term 35 (EL3204)
//     PlcTask Inputs/GVL_IO_REACTOR_CABINET.AI_10_R04S_HCoolingWaterPV <-> RTD Inputs Channel 1/Value
//     PlcTask Inputs/GVL_IO_REACTOR_CABINET.AI_10_Spare_02 <-> RTD Inputs Channel 2/Value
//     PlcTask Inputs/GVL_IO_REACTOR_CABINET.AI_10_Spare_03 <-> RTD Inputs Channel 3/Value
//     PlcTask Inputs/GVL_IO_REACTOR_CABINET.AI_10_Spare_04 <-> RTD Inputs Channel 4/Value
//   MU/MU Instance <-> Device 2 (EL6752)/SolValve
//     PlcTask Outputs/GVL_IO_VALVE.DO_00_V01ChalcogenCarrierChange <-> Connection (Poll)/Outputs/Output Data[0]
//     PlcTask Outputs/GVL_IO_VALVE.DO_00_V02MOCarreirChange <-> Connection (Poll)/Outputs/Output Data[0] @bit 1
//     PlcTask Outputs/GVL_IO_VALVE.DO_00_V03H2SeSourceChange <-> Connection (Poll)/Outputs/Output Data[0] @bit 2
//     PlcTask Outputs/GVL_IO_VALVE.DO_00_V04H2SSourceChange <-> Connection (Poll)/Outputs/Output Data[0] @bit 3
//     PlcTask Outputs/GVL_IO_VALVE.DO_00_V05Source_1TMInCarrierChange <-> Connection (Poll)/Outputs/Output Data[0] @bit 4
//     PlcTask Outputs/GVL_IO_VALVE.DO_00_V06Source_1TMInBypass <-> Connection (Poll)/Outputs/Output Data[0] @bit 5
//     PlcTask Outputs/GVL_IO_VALVE.DO_00_V07Source_2TMGaCarrierChange <-> Connection (Poll)/Outputs/Output Data[0] @bit 6
//     PlcTask Outputs/GVL_IO_VALVE.DO_00_V08Source_2TMGaBypass <-> Connection (Poll)/Outputs/Output Data[0] @bit 7
//     PlcTask Outputs/GVL_IO_VALVE.DO_00_V09Source_3DMSeCarrierChange <-> Connection (Poll)/Outputs/Output Data[1]
//     PlcTask Outputs/GVL_IO_VALVE.DO_00_V10Source_3DMSeBypass <-> Connection (Poll)/Outputs/Output Data[1] @bit 1
//     PlcTask Outputs/GVL_IO_VALVE.DO_00_V11Source_4ChalcogenCarrierChange <-> Connection (Poll)/Outputs/Output Data[1] @bit 2
//     PlcTask Outputs/GVL_IO_VALVE.DO_00_V12Source_4ChalcogenBypass <-> Connection (Poll)/Outputs/Output Data[1] @bit 3
//     PlcTask Outputs/GVL_IO_VALVE.DO_00_V13ReactorPurgeCarrierChange <-> Connection (Poll)/Outputs/Output Data[1] @bit 4
//     PlcTask Outputs/GVL_IO_VALVE.DO_00_V14Source_1TMInManifoldRun <-> Connection (Poll)/Outputs/Output Data[1] @bit 5
//     PlcTask Outputs/GVL_IO_VALVE.DO_00_V15Source_2TMGaManifoldRun <-> Connection (Poll)/Outputs/Output Data[1] @bit 6
//     PlcTask Outputs/GVL_IO_VALVE.DO_00_V16Source_3DMSeManifoldRun <-> Connection (Poll)/Outputs/Output Data[1] @bit 7
//     PlcTask Outputs/GVL_IO_VALVE.DO_00_V17GasH2SeManifoldRun <-> Connection (Poll)/Outputs/Output Data[2]
//     PlcTask Outputs/GVL_IO_VALVE.DO_00_V18GasH2SManifoldRun <-> Connection (Poll)/Outputs/Output Data[2] @bit 1
//     PlcTask Outputs/GVL_IO_VALVE.DO_00_V19Source_4ChalcogenManifoldRun <-> Connection (Poll)/Outputs/Output Data[2] @bit 2
//     PlcTask Outputs/GVL_IO_VALVE.DO_00_V20VentPress_Change <-> Connection (Poll)/Outputs/Output Data[2] @bit 3
//     PlcTask Outputs/GVL_IO_VALVE.DO_00_V21PumpByPass <-> Connection (Poll)/Outputs/Output Data[2] @bit 4
//     PlcTask Outputs/GVL_IO_VALVE.DO_00_V22DORVaccumON <-> Connection (Poll)/Outputs/Output Data[2] @bit 5
//     PlcTask Outputs/GVL_IO_VALVE.DO_00_V23DORFilling <-> Connection (Poll)/Outputs/Output Data[2] @bit 6
//     PlcTask Outputs/GVL_IO_VALVE.DO_00_V24Source_1LeakTest_IN <-> Connection (Poll)/Outputs/Output Data[2] @bit 7
//     PlcTask Outputs/GVL_IO_VALVE.DO_00_V26Source_2LeakTest_IN <-> Connection (Poll)/Outputs/Output Data[3] @bit 1
//     PlcTask Outputs/GVL_IO_VALVE.DO_00_V28Source_3LeakTest_IN <-> Connection (Poll)/Outputs/Output Data[3] @bit 3
//     PlcTask Outputs/GVL_IO_VALVE.DO_00_V30Source_4LeakTest_IN <-> Connection (Poll)/Outputs/Output Data[3] @bit 5
//     PlcTask Outputs/GVL_IO_VALVE.DO_00_V25Source_1LeakTest_OUT <-> Connection (Poll)/Outputs/Output Data[3]
//     PlcTask Outputs/GVL_IO_VALVE.DO_00_V27Source_2LeakTest_OUT <-> Connection (Poll)/Outputs/Output Data[3] @bit 2
//     PlcTask Outputs/GVL_IO_VALVE.DO_00_V29Source_3LeakTest_OUT <-> Connection (Poll)/Outputs/Output Data[3] @bit 4
//     PlcTask Outputs/GVL_IO_VALVE.DO_00_V31Source_4LeakTest_OUT <-> Connection (Poll)/Outputs/Output Data[3] @bit 6
//     PlcTask Outputs/GVL_IO_VALVE.DO_00_V32SourceVacuumON <-> Connection (Poll)/Outputs/Output Data[3] @bit 7
//   MU/MU Instance <-> Device 2 (EL6752)/TempController
//     PlcTask Inputs/GVL_DEVICE_NET_E3508.aInputActiveOut[1] <-> Connection (Poll)/Inputs/Input Data_5
//     PlcTask Inputs/GVL_DEVICE_NET_E3508.aInputActiveOut[2] <-> Connection (Poll)/Inputs/Input Data_6
//     PlcTask Inputs/GVL_DEVICE_NET_E3508.aInputAlarmStatus[1] <-> Connection (Poll)/Inputs/Input Data_7
//     PlcTask Inputs/GVL_DEVICE_NET_E3508.aInputAlarmStatus[2] <-> Connection (Poll)/Inputs/Input Data_8
//     PlcTask Inputs/GVL_DEVICE_NET_E3508.aInputDerivative[1] <-> Connection (Poll)/Inputs/Input Data_17
//     PlcTask Inputs/GVL_DEVICE_NET_E3508.aInputDerivative[2] <-> Connection (Poll)/Inputs/Input Data_18
//     PlcTask Inputs/GVL_DEVICE_NET_E3508.aInputIntegral[1] <-> Connection (Poll)/Inputs/Input Data_15
//     PlcTask Inputs/GVL_DEVICE_NET_E3508.aInputIntegral[2] <-> Connection (Poll)/Inputs/Input Data_16
//     PlcTask Inputs/GVL_DEVICE_NET_E3508.aInputManAutoBytes[1] <-> Connection (Poll)/Inputs/Input Data_9
//     PlcTask Inputs/GVL_DEVICE_NET_E3508.aInputManAutoBytes[2] <-> Connection (Poll)/Inputs/Input Data_10
//     PlcTask Inputs/GVL_DEVICE_NET_E3508.aInputPVBytes[1] <-> Connection (Poll)/Inputs/Input Data_1
//     PlcTask Inputs/GVL_DEVICE_NET_E3508.aInputPVBytes[2] <-> Connection (Poll)/Inputs/Input Data_2
//     PlcTask Inputs/GVL_DEVICE_NET_E3508.aInputProportional[1] <-> Connection (Poll)/Inputs/Input Data_13
//     PlcTask Inputs/GVL_DEVICE_NET_E3508.aInputProportional[2] <-> Connection (Poll)/Inputs/Input Data_14
//     PlcTask Inputs/GVL_DEVICE_NET_E3508.aInputSVBytes[1] <-> Connection (Poll)/Inputs/Input Data_3
//     PlcTask Inputs/GVL_DEVICE_NET_E3508.aInputSVBytes[2] <-> Connection (Poll)/Inputs/Input Data_4
//     PlcTask Inputs/GVL_DEVICE_NET_E3508.aInputStateAutoTune[1] <-> Connection (Poll)/Inputs/Input Data_11
//     PlcTask Inputs/GVL_DEVICE_NET_E3508.aInputStateAutoTune[2] <-> Connection (Poll)/Inputs/Input Data_12
//     PlcTask Outputs/GVL_DEVICE_NET_E3508.aOutputAlarmReset[1] <-> Connection (Poll)/Outputs/Output Data_7
//     PlcTask Outputs/GVL_DEVICE_NET_E3508.aOutputAlarmReset[2] <-> Connection (Poll)/Outputs/Output Data_8
//     PlcTask Outputs/GVL_DEVICE_NET_E3508.aOutputAutoTune_Enable[1] <-> Connection (Poll)/Outputs/Output Data_13
//     PlcTask Outputs/GVL_DEVICE_NET_E3508.aOutputAutoTune_Enable[2] <-> Connection (Poll)/Outputs/Output Data_14
//     PlcTask Outputs/GVL_DEVICE_NET_E3508.aOutputPowerBytes[1] <-> Connection (Poll)/Outputs/Output Data_5
//     PlcTask Outputs/GVL_DEVICE_NET_E3508.aOutputPowerBytes[2] <-> Connection (Poll)/Outputs/Output Data_6
//     PlcTask Outputs/GVL_DEVICE_NET_E3508.aOutputRate[1] <-> Connection (Poll)/Outputs/Output Data_11
//     PlcTask Outputs/GVL_DEVICE_NET_E3508.aOutputRate[2] <-> Connection (Poll)/Outputs/Output Data_12
//     PlcTask Outputs/GVL_DEVICE_NET_E3508.aOutputSVBytes[1] <-> Connection (Poll)/Outputs/Output Data_1
//     PlcTask Outputs/GVL_DEVICE_NET_E3508.aOutputSVBytes[2] <-> Connection (Poll)/Outputs/Output Data_2
//     PlcTask Outputs/GVL_DEVICE_NET_E3508.aOutputThreshold[1] <-> Connection (Poll)/Outputs/Output Data_9
//     PlcTask Outputs/GVL_DEVICE_NET_E3508.aOutputThreshold[2] <-> Connection (Poll)/Outputs/Output Data_10
//     PlcTask Outputs/GVL_DEVICE_NET_E3508.nOutputManAutoBytes[1] <-> Connection (Poll)/Outputs/Output Data_3
//     PlcTask Outputs/GVL_DEVICE_NET_E3508.nOutputManAutoBytes[2] <-> Connection (Poll)/Outputs/Output Data_4
//   MU/MU Instance <-> Device 2 (EL6752)/ThrottleValve
//     PlcTask Inputs/GVL_DEVICE_NET_IQ_PLUS.aInputPressurePV_CDG1[1] <-> Connection (Poll)/Inputs/Input 155_4
//     PlcTask Inputs/GVL_DEVICE_NET_IQ_PLUS.aInputPressurePV_CDG1[2] <-> Connection (Poll)/Inputs/Input 155_5
//     PlcTask Inputs/GVL_DEVICE_NET_IQ_PLUS.aInputPressurePV_CDG2[1] <-> Connection (Poll)/Inputs/Input 155_2
//     PlcTask Inputs/GVL_DEVICE_NET_IQ_PLUS.aInputPressurePV_CDG2[2] <-> Connection (Poll)/Inputs/Input 155_3
//     PlcTask Inputs/GVL_DEVICE_NET_IQ_PLUS.aInputPressureSP[1] <-> Connection (Poll)/Inputs/Input 155_6
//     PlcTask Inputs/GVL_DEVICE_NET_IQ_PLUS.aInputPressureSP[2] <-> Connection (Poll)/Inputs/Input 155_7
//     PlcTask Inputs/GVL_DEVICE_NET_IQ_PLUS.aInputValvePosionPV[1] <-> Connection (Poll)/Inputs/Input 155_8
//     PlcTask Inputs/GVL_DEVICE_NET_IQ_PLUS.aInputValvePosionPV[2] <-> Connection (Poll)/Inputs/Input 155_9
//     PlcTask Inputs/GVL_DEVICE_NET_IQ_PLUS.nInputStatus <-> Connection (Poll)/Inputs/Input 155_1
//     PlcTask Outputs/GVL_DEVICE_NET_IQ_PLUS.aOutputSVBytes[1] <-> Connection (Poll)/Outputs/Output 154[1]
//     PlcTask Outputs/GVL_DEVICE_NET_IQ_PLUS.aOutputSVBytes[2] <-> Connection (Poll)/Outputs/Output 154[2]
//     PlcTask Outputs/GVL_DEVICE_NET_IQ_PLUS.nOutputMode <-> Connection (Poll)/Outputs/Output 154[0]
//     PlcTask Outputs/GVL_DEVICE_NET_IQ_PLUS.nOutputSetType <-> Connection (Poll)/Outputs/Output 154[3]

// ---- DATA TYPES/E_ComState.TcDUT
TYPE E_ComState :
(
	IDLE,
	OPEN,
	CONNECTED,
	EXIST_MSG,
	SENDING,
	WAITING_RESPONSE,
	PARSING,
	CLOSING,
	ERROR
);
END_TYPE

// ---- DATA TYPES/E_MFC_INDEX.TcDUT
TYPE E_MFC_INDEX :
(
	MFC_CH_1,
	MFC_CH_2,
	MFC_CH_3,
	MFC_CH_4,
	MFC_CH_5,
	MFC_CH_6,
	MFC_CH_7,
	MFC_CH_8,
	MFC_CH_9,
	MFC_CH_10,
	MFC_CH_11
);
END_TYPE

// ---- DATA TYPES/MODUELS/ST_MAIN_MODULE.TcDUT
TYPE ST_MAIN_MODULE :
STRUCT

	TEMP_CONTROLLER:ST_TEMP_CONTROLLER;  // 구조가 변결 될 수  있음
	LINE_HEATER:ARRAY[1..8] OF ST_TEMP_CONTROLLER;// 구조가 변결 될 수  있음
	BATH_TEMP:ARRAY[1..3]OF ST_TEMP_CONTROLLER;
	THROTTLE_VALVE:ST_THROTTLE_VALVE;// 구조가 변결 될 수  있음
	ROTATION_MOTOR:ST_ROTATION_MOTOR; // jhkang_251112 추가됨
	UTILITY:ST_UTILITY;
END_STRUCT
END_TYPE

// ---- DATA TYPES/MODUELS/ST_NOTIFICATION.TcDUT
TYPE ST_NOTIFICATION :
STRUCT
	ENABLE:BOOL:=FALSE;
	RESET:BOOL:=TRUE;
	NOTIFICATION_TYPE:DINT; (* NOTIFI_INTERLOCK = 1, NOTIFI_ALARM = 2, NOTIFI_MESSAGE = 3 *)
	NOTIFICATION_ID:DINT;
	MESSAGE_BANK:ARRAY[1..40] OF ST_NOTIFICATION_MESSAGE;
	MESSAGE_BANK_COUNT:DINT;
END_STRUCT
END_TYPE

// ---- DATA TYPES/MODUELS/ST_REACTOR_CABINET.TcDUT
TYPE ST_REACTOR_CABINET :
STRUCT

	DI_01_MaintenanceModeKey :ST_DIGITAL_PART;
	DI_01_ReactorCabinetLampButton :ST_DIGITAL_PART;
	DI_01_DORVACButton :ST_DIGITAL_PART;
	DI_01_DORATMButton :ST_DIGITAL_PART;
	DI_01_ReactorDoorUpButton :ST_DIGITAL_PART;
	DI_01_ReactorDoorDownButton :ST_DIGITAL_PART;
	DI_01_ClampLock :ST_DIGITAL_PART;
	DI_01_ClampRelease :ST_DIGITAL_PART;
	
	DI_02_C_WFlowSensor :ST_DIGITAL_PART;
	DI_02_SusceptorRotationMotorFault :ST_DIGITAL_PART;
	DI_02_VacuumPumpFail :ST_DIGITAL_PART;
	DI_02_VacuumPumpWarning :ST_DIGITAL_PART;
	DI_02_VacuumPumpAlarm :ST_DIGITAL_PART;
	DI_02_VacuumPumpRunning :ST_DIGITAL_PART;
	DI_02_VacuumPumpFBRunning :ST_DIGITAL_PART;
	
	DI_02_ReactorDoorUpLimitSensor :ST_DIGITAL_PART;
	DI_03_ReactorDoorDownLimitSensor :ST_DIGITAL_PART;
	DI_03_CylinderAutoSwitch_Closed :ST_DIGITAL_PART;
	DI_03_CylinderAutoSwitch_Opened :ST_DIGITAL_PART;
	DI_03_ReactorCabinetDoorClose :ST_DIGITAL_PART;
	DI_03_Spare_01 :ST_DIGITAL_PART;
	DI_03_Spare_02 :ST_DIGITAL_PART;
	DI_03_Spare_03 :ST_DIGITAL_PART;
	DI_03_Spare_04 :ST_DIGITAL_PART;
	
	DO_04_SignalTowerRed :ST_DIGITAL_PART;
	DO_04_SignalTowerOrange :ST_DIGITAL_PART;
	DO_04_SignalTowerGreen :ST_DIGITAL_PART;
	DO_04_SignalTowerBlue :ST_DIGITAL_PART;
	DO_04_SignalTowerWhite :ST_DIGITAL_PART;
	DO_04_SignalTowerBuzzer :ST_DIGITAL_PART;
	DO_04_ReactorCoverUpRelay :ST_DIGITAL_PART;
	DO_04_ReactorCoverDownRelay :ST_DIGITAL_PART;
	
	DO_05_ClampLock :ST_DIGITAL_PART;
	DO_05_ClampRelease :ST_DIGITAL_PART;
	DO_05_VacuumPumpStart_Stop :ST_DIGITAL_PART;
	DO_05_VacuumPumpReset :ST_DIGITAL_PART;
	DO_05_SusceptorRotationFWD :ST_DIGITAL_PART;
	DO_05_SusceptorRotationSTOP :ST_DIGITAL_PART;
	DO_05_SusceptorRotationAL_RST :ST_DIGITAL_PART;
	DO_05_DORVACButtonLamp :ST_DIGITAL_PART;
	
	DO_06_DORATMButtonLamp :ST_DIGITAL_PART;
	DO_06_ReactorCoverUpButtonLamp :ST_DIGITAL_PART;
	DO_06_ReactorCoverDownButtonLamp :ST_DIGITAL_PART;
	DO_06_ClampLockButtonLamp :ST_DIGITAL_PART;
	DO_06_ClampReleaseButtonLamp :ST_DIGITAL_PART;
	DO_06_ReactorCabinetLamp :ST_DIGITAL_PART;
	DO_06_Spare07 :ST_DIGITAL_PART;
	DO_06_Spare08 :ST_DIGITAL_PART;
	
	AI_07_P02_ReactorPressure10TorrPV :ST_ANALOG_PART;
	AI_07_P03_ExhaustPressurePV :ST_ANALOG_PART;
	AI_07_S05_DORPressurePV :ST_ANALOG_PART;
	AI_07_Spare_04 :ST_ANALOG_PART;

	AI_08_R01SusceptorRotationPV :ST_ANALOG_PART;
	AI_08_Spare_02 :ST_ANALOG_PART;
	AI_08_Spare_03 :ST_ANALOG_PART;
	AI_08_Spare_04 :ST_ANALOG_PART;
	
	AO_09_P03_ExhaustPressureAM215Input :ST_ANALOG_PART;
	AO_09_R01_SusceptorRotationSV :ST_ANALOG_PART;
	AO_09_Spare_03 :ST_ANALOG_PART;
	AO_09_Spare_04 :ST_ANALOG_PART;
	
	AI_10_R04S_HCoolingWaterPV :ST_ANALOG_PART;
	AI_10_Spare_02 :ST_ANALOG_PART;
	AI_10_Spare_03 :ST_ANALOG_PART;
	AI_10_Spare_04 :ST_ANALOG_PART;
END_STRUCT
END_TYPE

// ---- DATA TYPES/MODUELS/ST_SEQUENCE.TcDUT
TYPE ST_SEQUENCE :
STRUCT
	SEQUENCE_1:ST_SEQUENCE_PART;
	SEQUENCE_2:ST_SEQUENCE_PART;
	SEQUENCE_3:ST_SEQUENCE_PART;
	SEQUENCE_4:ST_SEQUENCE_PART;
	SEQUENCE_5:ST_SEQUENCE_PART;
	SEQUENCE_6:ST_SEQUENCE_PART;
	SEQUENCE_7:ST_SEQUENCE_PART;
	SEQUENCE_8:ST_SEQUENCE_PART;
	SEQUENCE_9:ST_SEQUENCE_PART;
	SEQUENCE_10:ST_SEQUENCE_PART;
END_STRUCT
END_TYPE

// ---- DATA TYPES/MODUELS/ST_TEMP_CONTROLLER.TcDUT
TYPE ST_TEMP_CONTROLLER :
STRUCT
	CURRENT_MAN_AUTO:DINT;
	CURRENT_PV_TEMP:DINT;
	CURRENT_PV_POWER:DINT;
	CURRENT_PV_POWER_RATE:DINT;
	CURRENT_SET_VALUE:DINT;
	CURRENT_TARGET_VALUE:DINT;
	CURRENT_ACTIVE_OUT:DINT;
	CURRENT_ALARM_STATE:DINT;
	CURRENT_THRESHOLD:DINT;
	CURRENT_OUT:DINT;
	CURRENT_ALARM_CLEAR:DINT;
	
	SET_MANUAL_AUTO:DINT;
	SET_TEMP_SV:DINT;
	SET_TARGET_SET_POINT:DINT;
	SET_MANUAL_POWER:DINT;
	SET_HIGH_LIMIT:DINT;
	SET_ALARM_CLEAR:DINT;
END_STRUCT
END_TYPE

// ---- DATA TYPES/MODUELS/ST_THROTTLE_VALVE.TcDUT
TYPE ST_THROTTLE_VALVE :
STRUCT
	CURRENT_STATUS:DINT;
	CURRENT_CDG1_PRESSURE:DINT;(*1000Tor*)
	CURRENT_CDG2_PRESSURE:DINT;(*100Torr*)
	CURRENT_SET_PV:DINT;
	CURRENT_VALVE_POSITION:DINT;
	CURRENT_MODE:DINT;(*1: Pressure , 2:Position*)
	CURRENT_VALVE_MODE:DINT;
	
	SET_OUTPUT_MODE:DINT;
	SET_PRESSURE:DINT;
	SET_CONTROL_MODE:DINT;
	//1:Pressure Control, 2:Valve Position Control
END_STRUCT
END_TYPE

// ---- DATA TYPES/MODUELS/ST_UTILITY.TcDUT
TYPE ST_UTILITY :
STRUCT
	TOTAL_FLOW_CAL:DINT;
	TOTAL_FLOW_MO:DINT;
	SPARE_1:DINT;
	SPARE_2:DINT;
	SPARE_3:DINT;
	SPARE_4:DINT;
	SPARE_5:DINT;
	SPARE_6:DINT;
	SPARE_7:DINT;
	SPARE_8:DINT;
	SPARE_9:DINT;
	SPARE_10:DINT;
END_STRUCT
END_TYPE

// ---- DATA TYPES/MODUELS/ST_ROTATION_MOTOR.TcDUT
TYPE ST_ROTATION_MOTOR :
STRUCT
	CURRENT_STATUS:DINT;
	CURRENT_PV:REAL;
	CURRENT_SET_PV:DINT;
	
	SET_CONTROL_VALUE:REAL;
	SET_PRESSURE:DINT;
	SET_CONTROL_MODE:DINT;
END_STRUCT
END_TYPE

// ---- DATA TYPES/PARTS/ST_ANALOG_PART.TcDUT
TYPE ST_ANALOG_PART :
STRUCT
	PART_ID:DINT;
	VALUE:LREAL;
	SPARE:DINT;
END_STRUCT
END_TYPE

// ---- DATA TYPES/PARTS/ST_DIGITAL_PART.TcDUT
TYPE ST_DIGITAL_PART :
STRUCT
	PART_ID:DINT;
	VALUE:BOOL;
	UI_NUMBER:DINT;
END_STRUCT
END_TYPE

// ---- DATA TYPES/PARTS/ST_SEQUENCE_PART.TcDUT
TYPE ST_SEQUENCE_PART :
STRUCT
	PARTID:DINT;
	STATUS:DINT;
	CURRENT_STEP:DINT;
	MESSAGE: STRING(100);
END_STRUCT
END_TYPE

// ---- DEVICE/ST_LineHeater_Data.TcDUT
TYPE ST_LineHeater_Data :
STRUCT
	LINE_HEATER_CH_1_PV_VALUE:WORD;(*1*)
	LINE_HEATER_CH_1_DOT:WORD;(*2*)
	LINE_HEATER_CH_1_UNIT:WORD;(*3*)
	LINE_HEATER_CH_1_SETVALUE:WORD;(*4*)
	LINE_HEATER_CH_1_HEATING_MV:WORD;(*5*)
	LINE_HEATER_CH_1_COOLING_MV:WORD;(*6*)
	
	LINE_HEATER_CH_2_PV_VALUE:WORD;(*1*)
	LINE_HEATER_CH_2_DOT:WORD;(*2*)
	LINE_HEATER_CH_2_UNIT:WORD;(*3*)
	LINE_HEATER_CH_2_SETVALUE:WORD;(*4*)
	LINE_HEATER_CH_2_HEATING_MV:WORD;(*5*)
	LINE_HEATER_CH_2_COOLING_MV:WORD;(*6*)
	
	LINE_HEATER_CH_3_PV_VALUE:WORD;(*1*)
	LINE_HEATER_CH_3_DOT:WORD;(*2*)
	LINE_HEATER_CH_3_UNIT:WORD;(*3*)
	LINE_HEATER_CH_3_SETVALUE:WORD;(*4*)
	LINE_HEATER_CH_3_HEATING_MV:WORD;(*5*)
	LINE_HEATER_CH_3_COOLING_MV:WORD;(*6*)
	
	LINE_HEATER_CH_4_PV_VALUE:WORD;(*1*)
	LINE_HEATER_CH_4_DOT:WORD;(*2*)
	LINE_HEATER_CH_4_UNIT:WORD;(*3*)
	LINE_HEATER_CH_4_SETVALUE:WORD;(*4*)
	LINE_HEATER_CH_4_HEATING_MV:WORD;(*5*)
	LINE_HEATER_CH_4_COOLING_MV:WORD;(*6*)
END_STRUCT
END_TYPE

// ---- DEVICE/ST_Modbus_Send_Frame.TcDUT
TYPE ST_Modbus_Send_Frame :
STRUCT
	UnitID:BYTE;
	StartAddress		:WORD;
	sendQuantity		:WORD;
	SendData			:ARRAY [0..10] OF WORD;
END_STRUCT
END_TYPE

// ---- DUTs/AnalogController.TcDUT
TYPE AnalogController :
STRUCT
	pv : REAL;
	
	cvController : FB_ControlRampGenerator;
END_STRUCT
END_TYPE

// ---- DUTs/DUTs/ENUM/E_aAnalogInputIO_Index.TcDUT
{attribute 'qualified_only'}
{attribute 'strict'}
{attribute 'to_string'}
TYPE E_aAnalogInputIO_Index :
(
	E_PV_MFC_01 :=1,
	E_PV_MFC_02 :=2,
	E_PV_MFC_03 :=3,
	E_PV_MFC_04 :=4,
	E_PV_MFC_05 :=5,
	E_PV_MFC_06 :=6,
	E_PV_MFC_07 :=7,
	E_PV_MFC_08 :=8,
	E_PV_MFC_09 :=9,
	E_PV_MFC_10 :=10,
	E_PV_MFC_11 :=11,
	E_PV_EPC_01 :=12,
	E_PV_Susceptor_Temp:=13,
	E_PV_Reactor_Pressure:=14,
	E_PV_susceptorRotation:=15,
	E_PV_Ultimate_Pressure:=20,
	E_PV_Exhaust_Pressure:=21,
	E_PV_DOR_PRESSURE:=22,
	E_PV_GAS_Pressure_N2:=23,
	E_PV_GAS_Pressure_H2:=24,
	E_PV_GAS_Pressure_H2S:=25,
	E_PV_GAS_Pressure_H2Se:=26,
	E_PV_CoolingWafer_SH:=27
);
END_TYPE

// ---- DUTs/DUTs/ENUM/E_AlarmList.TcDUT
{attribute 'qualified_only'}
{attribute 'strict'}
{attribute 'to_string'}
TYPE E_AlarmList :
(
	E_AlarmList_GasPressure_Low_N2:=1,
	E_AlarmList_GasPressureLowN2,
	E_AlarmList_GasPressureLowH2,
	E_AlarmList_GasPressureLowNH3,
	E_AlarmList_GasPressureLowSiH4,
	E_AlarmList_CWTemperatureHighSH,
	E_AlarmList_CWTemperatureHighCoil,
	E_AlarmList_SusceptorOverTemperature,
	E_AlarmList_ReactorOverPressure,
	E_AlarmList_PneumaticPressureLow,
	E_AlarmList_CoolingWaterLow,
	E_AlarmList_InductionHeaterFault,
	E_AlarmList_RotationMotorFault,
	E_AlarmList_VacuumPumpFault,
	E_AlarmList_GasCabinetDoorOpen,
	E_AlarmList_ReactorCabinetDoorOpen,
	E_AlarmList_SusceptorTemperatureDeviation,
	E_AlarmList_ReactorPressureDeviation,
	E_AlarmList_SusceptorRotationDeviation,
	E_AlarmList_MORunDeviation,
	E_AlarmList_HydRunDeviation,
	E_AlarmList_NH3LargeINDeviation,
	E_AlarmList_NH3SmallINDeviation,
	E_AlarmList_SiHINDeviation,
	E_AlarmList_SiHDilutionDeviation,
	E_AlarmList_SiHDilutedDeviation,
	E_AlarmList_TEBBubblingDeviation,
	E_AlarmList_TMAlBubblingDeviation,
	E_AlarmList_TMInBubblingDeviation,
	E_AlarmList_TMGaBubblingDeviation,
	E_AlarmList_DTMGaBubblingDeviation,
	E_AlarmList_DTMGaDilutionDeviation,
	E_AlarmList_DTMGaDilutedDeviation,
	E_AlarmList_Cp2MgBubblingDeviation,
	E_AlarmList_ReactorPurgeDeviation,
	E_AlarmList_RotationSealPurgeDeviation,
	E_AlarmList_MOVentDeviation,
	E_AlarmList_HydVentDeviation,
	E_AlarmList_SiH4PressureDeviation,
	E_AlarmList_TEBPressureDeviation,
	E_AlarmList_TMAlPressureDeviation,
	E_AlarmList_TMInPressureDeviation,
	E_AlarmList_TMGaPressureDeviation,
	E_AlarmList_DTMGaPressureDeviation,
	E_AlarmList_Cp2MgPressureDeviation,
	E_AlarmList_END

);
END_TYPE

// ---- DUTs/DUTs/ENUM/E_InputState.TcDUT
{attribute 'qualified_only'}
{attribute 'strict'}
{attribute 'to_string'}
TYPE E_InputState :
(
	E_Input_MaintKey,
	Reactor_Cabinet_Lamp,
	Gas_Cabinet_Lamp,
	PowerDistribute_Lamp,
	AirPressure_Sensor,
	WaferFlow_Sensor,
	E3508_Heater_Ready,
	E3508_Heater_Run,
	E3508_Heater_Fault,
	Rotation_Start,
	Rotation_Break,
	Rotation_Fault,
	Pump_Warning,
	Pump_running,
	Pump_Fault,
	Reactor_Cabinet_Door,
	Gas_Cabinet_Door,
	PowerDistri_Cabinet_Door,
	
	E_InputState_END

);
END_TYPE

// ---- DUTs/DUTs/ENUM/E_Interlock.TcDUT
{attribute 'qualified_only'}
{attribute 'strict'}
{attribute 'to_string'}
TYPE E_Interlock :
(
	AlarmTrig,
	WarningTrig,
	N2PressureLowAlarm,
	N2PressureLowWaring,
	H2PressureLowAlarm,
	H2PressureLowWarning,
	NH3PressureLowAlarm,
	NH2PressureLowWaring,
	SiH4PressureLowAlarm,
	SiH4PressureLowWarning,
	RecipeStartEnable,
	ReactorOpenEnable,
	HeatercanbeturnON,
	PumpcanbeturnON,  // GVL_IO.aInterlock[1].13
	
	ALARM_POPUP_GasPressureLowN2,
	ALARM_POPUP_GasPressureLowH2,
	ALARM_POPUP_GasPressureLowNH3,
	ALARM_POPUP_GasPressureLowSiH4,
	ALARM_POPUP_CWTemperatureHighSH,
	ALARM_POPUP_CWTemperatureHighCoil,
	ALARM_POPUP_SusceptorOverTemperature,
	ALARM_POPUP_ReactorOverPressure,
	ALARM_POPUP_PneumaticPressureLow,
	ALARM_POPUP_CoolingWaterLow,
	ALARM_POPUP_InductionHeaterFault,
	ALARM_POPUP_RotationMotorFault,
	ALARM_POPUP_VacuumPumpFault,
	ALARM_POPUP_GasCabinetDoorOpen,
	ALARM_POPUP_ReactorCabinetDoorOpen,
	ALARM_POPUP_SusceptorTemperatureDeviation,
	ALARM_POPUP_ReactorPressureDeviation,
	ALARM_POPUP_SusceptorRotationDeviation,
	ALARM_POPUP_MORunDeviation,
	ALARM_POPUP_HydRunDeviation,
	ALARM_POPUP_NH3LargeINDeviation,
	ALARM_POPUP_NH3SmallINDeviation,
	ALARM_POPUP_SiHINDeviation,
	ALARM_POPUP_SiHDilutionDeviation,
	ALARM_POPUP_SiHDilutedDeviation,
	ALARM_POPUP_TEBBubblingDeviation,
	ALARM_POPUP_TMAlBubblingDeviation,
	ALARM_POPUP_TMInBubblingDeviation,
	ALARM_POPUP_TMGaBubblingDeviation,
	ALARM_POPUP_DTMGaBubblingDeviation,
	ALARM_POPUP_DTMGaDilutionDeviation,
	ALARM_POPUP_DTMGaDilutedDeviation,
	ALARM_POPUP_Cp2MgBubblingDeviation,
	ALARM_POPUP_ReactorPurgeDeviation,
	ALARM_POPUP_RotationSealPurgeDeviation,
	ALARM_POPUP_MOVentDeviation,
	ALARM_POPUP_HydVentDeviation,
	ALARM_POPUP_SiH4PressureDeviation,
	ALARM_POPUP_TEBPressureDeviation,
	ALARM_POPUP_TMAlPressureDeviation,
	ALARM_POPUP_TMInPressureDeviation,
	ALARM_POPUP_TMGaPressureDeviation,
	ALARM_POPUP_DTMGaPressureDeviation,
	ALARM_POPUP_Cp2MgPressureDeviation,
	WARNING_POPUP_GasPressureLowN2,
	WARNING_POPUP_GasPressureLowH2,
	WARNING_POPUP_GasPressureLowNH3,
	WARNING_POPUP_GasPressureLowSiH4,
	WARNING_POPUP_CWTemperatureHighSH,
	WARNING_POPUP_CWTemperatureHighCoil,
	WARNING_POPUP_SusceptorOverTemperature,
	WARNING_POPUP_ReactorOverPressure,
	WARNING_POPUP_PneumaticPressureLow,
	WARNING_POPUP_CoolingWaterLow,
	WARNING_POPUP_InductionHeaterFault,
	WARNING_POPUP_RotationMotorFault,
	WARNING_POPUP_VacuumPumpFault,
	WARNING_POPUP_GasCabinetDoorOpen,
	WARNING_POPUP_ReactorCabinetDoorOpen,
	WARNING_POPUP_SusceptorTemperatureDeviation,
	WARNING_POPUP_ReactorPressureDeviation,
	WARNING_POPUP_SusceptorRotationDeviation,
	WARNING_POPUP_MORunDeviation,
	WARNING_POPUP_HydRunDeviation,
	WARNING_POPUP_NH3LargeINDeviation,
	WARNING_POPUP_NH3SmallINDeviation,
	WARNING_POPUP_SiHINDeviation,
	WARNING_POPUP_SiHDilutionDeviation,
	WARNING_POPUP_SiHDilutedDeviation,
	WARNING_POPUP_TEBBubblingDeviation,
	WARNING_POPUP_TMAlBubblingDeviation,
	WARNING_POPUP_TMInBubblingDeviation,
	WARNING_POPUP_TMGaBubblingDeviation,
	WARNING_POPUP_DTMGaBubblingDeviation,
	WARNING_POPUP_DTMGaDilutionDeviation,
	WARNING_POPUP_DTMGaDilutedDeviation,
	WARNING_POPUP_Cp2MgBubblingDeviation,
	WARNING_POPUP_ReactorPurgeDeviation,
	WARNING_POPUP_RotationSealPurgeDeviation,
	WARNING_POPUP_MOVentDeviation,
	WARNING_POPUP_HydVentDeviation,
	WARNING_POPUP_SiH4PressureDeviation,
	WARNING_POPUP_TEBPressureDeviation,
	WARNING_POPUP_TMAlPressureDeviation,
	WARNING_POPUP_TMInPressureDeviation,
	WARNING_POPUP_TMGaPressureDeviation,
	WARNING_POPUP_DTMGaPressureDeviation,
	WARNING_POPUP_Cp2MgPressureDeviation,
	E_Interlock_END
);
END_TYPE

// ---- DUTs/DUTs/ENUM/E_Morning_Index.TcDUT
{attribute 'qualified_only'}
{attribute 'strict'}
{attribute 'to_string'}
TYPE E_Morning_Index :
(
	E_Morning_UltimatePressure:=1,
	E_Morning_ExhaustPressure:=2,
	E_Morning_DoubleOring:=3,
	E_Morning_GasPressure_N2:=4,
	E_Morning_GasPressure_H2:=5,
	E_Morning_GasPressure_H2S:=6,
	E_Morning_GasPressure_H2SE:=7,
	E_Morning_CoolingWafer_SH:=8,
	E_Morning_DP_Chalcogen:=9,
	E_Morning_MO_DP:=10,
	E_Morning_TempPowerRate:=11,
	E_Morning_TV_Position:=12,
	E_Morning_TB_Temp_1:=13,
	E_Morning_TB_Temp_2:=14,
	E_Morning_TB_Temp_3:=15,
	E_Morning_TB_Temp_4:=16,
	E_Morning_Total_Flow_MOD:=17,
	E_Morning_Total_Flow_HYD:=18
);
END_TYPE

// ---- DUTs/DUTs/F_GetReal_USINT.TcDUT
TYPE F_GetReal_USINT :
UNION
	Input_USINT : ARRAY[1..2]OF USINT;
	Output_Real:REAL;
END_UNION
END_TYPE

// ---- DUTs/GeneralIO.TcDUT
TYPE GeneralIO :
STRUCT
	control: ARRAY [1..GVL_CONSTANT.NumGeneralIOControl] OF BYTE;
	state: ARRAY [1..GVL_CONSTANT.NumGeneralIOState] OF BYTE;
END_STRUCT
END_TYPE

// ---- DUTs/Interlock/Interlock.TcDUT
TYPE Interlock :
STRUCT
	interlockSetting : InterlockSetting;
	interlockState : InterlockState;
	Interlock_Return_Message :T_MaxString;  (*plc에서 특정 Trig를 True로 바꾸면 UI에서는 이 메시지를 Popup ??   *)
END_STRUCT
END_TYPE

// ---- DUTs/Interlock/InterlockEnableThreshold.TcDUT
TYPE InterlockEnableThreshold :
STRUCT
	enable : BOOL;
	threshold : REAL;
END_STRUCT
END_TYPE

// ---- DUTs/Interlock/InterlockSetting.TcDUT
TYPE InterlockSetting :
STRUCT
	aInterlockEnableThreshold	: ARRAY[1..GVL_CONSTANT.NumInterlockSettingEnableThreshold] OF InterlockEnableThreshold;
	aInterlockEnable : ARRAY[1..GVL_CONSTANT.NumInterlockSettingEnable] OF BOOL;
	
	aAnalogAlarmEnable		: ARRAY[1..GVL_CONSTANT.NumInterlockSettingAnalogEnable] OF BOOL; 
	aAnalogWarningEnable		: ARRAY[1..GVL_CONSTANT.NumInterlockSettingAnalogEnable] OF BOOL; 
	aDigitalAlarmEnable		: ARRAY[1..GVL_CONSTANT.NumInterlockSettingDigitalEnable] OF BOOL; 
	aDigitalWarningEnable		: ARRAY[1..GVL_CONSTANT.NumInterlockSettingDigitalEnable] OF BOOL; 
END_STRUCT
END_TYPE

// ---- DUTs/Interlock/InterlockState.TcDUT
TYPE InterlockState :
STRUCT
	aLogicalInterlock				: ARRAY[1..GVL_CONSTANT.NumLogicalInterlockState] OF BOOL;
	aInterlockSubstate				: LogicalInterlockSubstate;
	aAlarmState						: ARRAY[1..GVL_CONSTANT.NumInterlockAlarmWarningState] OF BOOL;
	aWarningState					: ARRAY[1..GVL_CONSTANT.NumInterlockAlarmWarningState] OF BOOL;
END_STRUCT
END_TYPE

// ---- DUTs/Interlock/LogicalInterlockSubstate.TcDUT
TYPE LogicalInterlockSubstate :
STRUCT
	recipeEnableSubstate : ARRAY[1..GVL_CONSTANT.NumInterlockRecipeEnableSubstate] OF BOOL;
	openReactorSubstate : ARRAY[1..GVL_CONSTANT.NumInterlockOpenReactorSubstate] OF BOOL;
END_STRUCT
END_TYPE

// ---- DUTs/IO/AnalogIO.TcDUT
TYPE AnalogIO :
STRUCT
	(* Analog Input to INT*)
	aAnalogInputIO 	: ARRAY[1..GVL_CONSTANT.NumAnalogInput] OF INT;
	aAnalogOutputIO : ARRAY[1..GVL_CONSTANT.NumAnalogOutput] OF INT;
END_STRUCT
END_TYPE

// ---- DUTs/IO/DigitalIO.TcDUT
TYPE DigitalIO :
STRUCT
	(* Digital IO to Byte *)
	aDigitalInputIO 	: ARRAY[1..GVL_CONSTANT.NumDigitalInput] OF BOOL; //KL1408 9EA
	aDigitalOutputIO : ARRAY[1..GVL_CONSTANT.NumDigitalOutput] OF BOOL; //KL2408 4EA
END_STRUCT
END_TYPE

// ---- DUTs/IO/IO.TcDUT
TYPE IO :
STRUCT
	digital: DigitalIO;
	analog: AnalogIO;
END_STRUCT
END_TYPE

// ---- DUTs/MainPRGControl.TcDUT
TYPE MainPRGControl :
STRUCT
	controlModeCmd : E_ControlMode := E_ControlMode.Manual;
	controlMode	: E_ControlMode := controlModeCmd;
END_STRUCT
END_TYPE

// ---- DUTs/Recipe/Recipe.TcDUT
TYPE Recipe :
STRUCT
	aRecipe		: ARRAY[1..GVL_CONSTANT.MaxRecipeStep] OF RecipeStep; //Recipe Structure
	iRcpTotalStep			: INT; //Recip Total Number
	control : RecipeControl;
END_STRUCT
END_TYPE

// ---- DUTs/Recipe/RecipeControl.TcDUT
TYPE RecipeControl :
STRUCT
	iRcpStepN				: INT;
	cmd_RcpOperation		: INT; // 0:Inital State, 10:RUN, 20:PAUSE, 30:RESTART, 40:STOP, 60:SKIP, 90:ManualOperation
	userState				: INT;	// 0:Inital State, 10:RUN, 20:PAUSE, 30:RESTART, 40:STOP, 50:END, 60:SKIP
	
	Pause_ET				: TIME := T#0S;
	RecipeRunET 			: RecipeRunET; 
END_STRUCT
END_TYPE

// ---- DUTs/Recipe/RecipeStep.TcDUT
TYPE RecipeStep :
STRUCT
	sRecipe : STRING(GVL_CONSTANT.MaxRecipeNameLength);
	iRecipe : ARRAY[1..GVL_CONSTANT.RecipeNumReactorCondition] OF INT; //Reactor Condition
	rRecipe : ARRAY[1..GVL_CONSTANT.NumAnalogController] OF REAL; //MFC, EPC Data
	cTemp 	: REAL := 0; 	
	dRecipe : DWORD; //Valve Data
END_STRUCT
END_TYPE

// ---- DUTs/Recipe/ScaleFactor.TcDUT
TYPE ScaleFactor :
STRUCT
	MinFactor	: USINT; // Sensor Minimum Range
	MaxFactor	: USINT; // Sensor Maximum Range
END_STRUCT
END_TYPE

// ---- GVLs/GVL_INTERFACE_UI.TcGVL
{attribute 'qualified_only'}
VAR_GLOBAL
	aOutputSolValve 		: ARRAY[1..GVL_CONSTANT.NumSolValve] OF BOOL; //Solenoid Valve
	aAnalogController 		: ARRAY[1..GVL_CONSTANT.NumAnalogController] OF AnalogController; //Flow Controller (Ramp Controller) for MFC, EPC, Reactor
	aMaxValue		: ARRAY[1..GVL_CONSTANT.NumAnalogController] OF REAL; //Max Value set from UI Application
	
	(* Present Value Meter Display*)
	aMonitoring_PV 			: ARRAY[1..GVL_CONSTANT.NumMonitoring] OF REAL; //Gauge Monitoring Value to UI
	
	interlock 				: Interlock;
	generalIO				: GeneralIO;
	mainPRGControl : MainPRGControl;
	recipe :Recipe;
END_VAR

// ---- GVLs/GVL_CONSTANT.TcGVL
{attribute 'qualified_only'}
VAR_GLOBAL CONSTANT
	MFC_SEND_CYCLE_TIME:TIME :=T#200MS;
	
	EL3064MaxValueH	: REAL := 16383; //0~5V Half Input
	EL3064MaxValue 	: REAL := 32767; //0~10V
	EL4004MaxValueH	: REAL := 16383; //0~5V Half Output
	EL4004MaxValue 	: REAL := 32767; //4~20mA
	EL3102MAxValue	: REAL := 32767;
	
	NumAnalogController : UINT := 15;
	NumFlowController : UINT := 12;
	NumReactor : UINT := NumAnalogController - NumFlowController;
	
	NumAnalogInput : UINT := 40;
	NumAnalogOutput : UINT := 42;
	NumDigitalInput : UINT := 80; //jhkang Spare 포함
	NumDigitalOutput : UINT := 50;//jhkang Spare 포함
	
	NumGeneralIOControl : UINT := 11;
	NumGeneralIOState : UINT := 100;
	
	NumInterlockSettingEnable : UINT := 9;
	NumInterlockSettingEnableThreshold : UINT := 12;
	NumInterlockSettingDigitalEnable : UINT := 20;
	NumInterlockSettingAnalogEnable : UINT := 20;
	
	NumLogicalInterlockState : UINT := 20;
	NumInterlockAlarmWarningState : UINT := 40;
	NumInterlockRecipeEnableSubstate : UINT := 11;
	NumInterlockOpenReactorSubstate : UINT := 12;
	
	NumSolValve : UINT := 28;
	NumMonitoring : UINT := 15;
	
	MaxRecipeStep : UINT := 100;
	MaxRecipeNameLength : UINT := 81;
	RecipeNumReactorCondition : UINT := 5;
	
	cSTX : BYTE := 16#02;
	cETX : BYTE := 16#03;
END_VAR

// ---- GVLs/GVL_DEVICE_NET_E3508.TcGVL
{attribute 'qualified_only'}
VAR_GLOBAL
	(*E3508*)
	(*Input*)
	aInputPVBytes 			AT %I*: ARRAY[1..2]OF USINT; //Loop1 PV
	aInputSVBytes 			AT %I*: ARRAY[1..2]OF USINT; //Loop1 Working PV
	aInputActiveOut 		AT %I*: ARRAY[1..2]OF USINT; //Loop1 Main.ActiveOut
	aInputAlarmStatus 		AT %I*: ARRAY[1..2]OF USINT; //Alarm status
	aInputManAutoBytes 		AT %I*: ARRAY[1..2]OF USINT; // Loop1 Main.AutoMan
	aInputStateAutoTune		AT %I*: ARRAY[1..2]OF USINT; // Loop1 State Auto Tune
	aInputProportional			AT %I*: ARRAY[1..2]OF USINT; // Loop1 State Auto Tune
	aInputIntegral			AT %I*: ARRAY[1..2]OF USINT; // Loop1 State Auto Tune
	aInputDerivative			AT %I*: ARRAY[1..2]OF USINT; // Loop1 State Auto Tune
	
//	aInputAlarmThreshold 	AT %I*: ARRAY[1..2]OF USINT; //Alarm1 Threshold
//	aInputAlarmOut 			AT %I*: ARRAY[1..2]OF USINT; //Alarm.1.Out
//	aInputAlarmSummary 		AT %I*: ARRAY[1..2]OF USINT; // AlmSummary.AnyAlarm (Alarm Clear)

	(*Output*)
	aOutputSVBytes 			AT %Q*: ARRAY[1..2]OF USINT; //Loop.1.Main.TagetSP
	nOutputManAutoBytes 	AT %Q*: ARRAY[1..2]OF USINT; //Loop.1.Main.AutoMan
	aOutputPowerBytes 	AT %Q*: ARRAY[1..2]OF USINT; //Loop1 OP.ManualOutVal
	aOutputAlarmReset	 	AT %Q*: ARRAY[1..2]OF USINT; //Loop1 Alarm Reset
	aOutputThreshold 		AT %Q*: ARRAY[1..2]OF USINT; //Alarm.1.Threshold
	aOutputRate 		AT %Q*: ARRAY[1..2]OF USINT; //Rate
	aOutputAutoTune_Enable 		AT %Q*: ARRAY[1..2]OF USINT; //Auto Tune
	
END_VAR


//EUROTHERM input
//1 PV1  
//2 PV2
//3 SV1
//4 SV2   / 10
//5 Active Out /10
//6 Active Out /10
//7 alarm
//8 alarm
//9  manual auto
//10 manual auto
//11 PID STATUE
//12 PID STATUE
//13 PID p / 10
//14 PID p / 10 
//15 PID I 360
//16 PID I 360
//17 PID D 60
//18 PID D 60

// ---- GVLs/GVL_DEVICE_NET_IQ_PLUS.TcGVL
{attribute 'qualified_only'}
VAR_GLOBAL
	(*IQ PLUS*)
	(*Input*)
	nInputStatus AT %I* : USINT; //Input Status Bytes
	aInputPressurePV_CDG2 AT %I* : ARRAY[1..2]OF USINT; //CDG2 Pressure
	aInputPressurePV_CDG1 AT %I* : ARRAY[1..2]OF USINT; //CDG1 Pressure
	aInputPressureSP AT %I* : ARRAY[1..2]OF USINT; //Set Point Pressure
	aInputValvePosionPV AT %I* : ARRAY[1..2]OF USINT; //Current Valve Position
	
	(*Output*)
	//Output to IQ-PLUS Throttle Valve
	nOutputMode AT %Q* : USINT;//0 : normal 1:Close , 2:Open Valve , 3:Hold , 4:Reset
	aOutputSVBytes AT %Q* : ARRAY[1..2]OF USINT; //Set Pressure
	nOutputSetType AT %Q* : USINT; //1:Pressure Control, 2:Valve Position Control
	
END_VAR

// ---- GVLs/GVL_IO.TcGVL
{attribute 'qualified_only'}
VAR_GLOBAL
	io : IO;
	ControlDevice :ST_MAIN_MODULE;
	
//// 	nCaseSignalTower		: INT;
//// 	nDorOperationError		: INT;
//// 	bDorState				: BOOL;
//// 	bDorOnEnable			: BOOL;
//// //bE3508_HeaterOn			: BOOL;
//// 	wE3508_CV				: WORD;
//// 	wE3508_PV				: WORD;
//// 	wIqPlus_CV				: WORD;
//// 	wIqPlus_CDG1_PV			: WORD;
//// 	wIqPlus_CDG2_PV			: WORD;
//// 	nRotation_Converted_PV	: REAL;
//// 	rRotation_ControlValue	: REAL;
//// 	nIQPLUS_SetType 		: INT;
//// 	nIQPLUS_Mode			: INT;
//// 	aLineHeater_rTemperaturePV : ARRAY[1..8]OF REAL;
//// 	nE3508_nInputManAutoBytes : USINT;
//// 	isCoverClosed 			: BOOL;
//// 	isPumpRunning 			: BOOL;
//// 	
//// 	UI_INTERLOCK_CHECK_RECIPE_ENABLE:WORD;(**)
//// 	UI_INTERLOCK_CHECK_OPEN_REACTOR:WORD;(**)
	nRotation_Converted_PV: INT;
END_VAR

// ---- GVLs/GVL.TcGVL
{attribute 'qualified_only'}
VAR_GLOBAL
	MainModule:ST_MAIN_MODULE;
	fbLineHeater_Manager:FB_LINE_HEATER_MANAGER;
	
	RotationResetTon: TON;
	
	Horiba_Mfc : ARRAY[1..10] OF ST_MfcData := [
											(Addr:='@01'),(Addr:='@02'),(Addr:='@03'),(Addr:='@04'),(Addr:='@05'),
											(Addr:='@06'),(Addr:='@07'),(Addr:='@08'),(Addr:='@09'),(Addr:='@0A')];
END_VAR

// ---- GVLs/GVL_IO_GAS_CABINET.TcGVL
{attribute 'qualified_only'}
VAR_GLOBAL
	DI_01_ResetButton AT%I*:BOOL;
	DI_01_GasCabinetLampButton AT%I*:BOOL;
	DI_01_PneumaticPressureSensor AT%I*:BOOL;
	DI_01_GasCabinetDoorClose AT%I*:BOOL;
	DI_01_ControlCabinetDoorClose AT%I*:BOOL;
	DI_01_SMPS_1Alarm AT%I*:BOOL;
	DI_01_SMPS_2Alarm AT%I*:BOOL;
	DI_01_SMPS_3Alarm AT%I*:BOOL;
	
	DI_02_SMPS_4Alarm AT%I*:BOOL;
	DI_02_GraphiteHeaterELCB AT%I*:BOOL;
	DI_02_ThermalBathsELCB AT%I*:BOOL;
	DI_02_VacuumPumpELCB AT%I*:BOOL;
	DI_02_LineHeatersELCB AT%I*:BOOL;
	DI_02_RotationMotorCP AT%I*:BOOL;
	DI_02_CoverLiftMotorCP AT%I*:BOOL;
	DI_02_T_VCP AT%I*:BOOL;
	
	DI_03_GasDetectorCP AT%I*:BOOL;
	DI_03_CabinetLampsCP AT%I*:BOOL;
	DI_03_MFCPowerCP AT%I*:BOOL;
	DI_03_LineHeater_1CP AT%I*:BOOL;
	DI_03_LineHeater_2CP AT%I*:BOOL;
	DI_03_LineHeater_3CP AT%I*:BOOL;
	
	DI_03_LineHeater_4CP AT%I*:BOOL;
	DI_03_LineHeater_5CP AT%I*:BOOL;
	DI_04_LineHeater_6CP AT%I*:BOOL;
	DI_04_LineHeater_7CP AT%I*:BOOL;
	DI_04_LineHeater_8CP AT%I*:BOOL;
	DI_04_GasDetectorH2 AT%I*:BOOL;
	DI_04_GasDetectorH2S AT%I*:BOOL;
	DI_04_GasDetectorH2Se AT%I*:BOOL;
	DI_04_FireSensor AT%I*:BOOL;
	DI_04_ExternalScrubberFault AT%I*:BOOL;
	
	DI_05_ExternalH2GasCabinetFault AT%I*:BOOL;
	DI_05_ExternalH2SGasCabinetFault AT%I*:BOOL;
	DI_05_ExternalH2SeGasCabinetFault AT%I*:BOOL;
	DI_05_ExternalUserInputAlarm AT%I*:BOOL;
	DI_05_ThermalBath_1DeviationAlarm AT%I*:BOOL;
	DI_05_ThermalBath_1CutOffAlarm AT%I*:BOOL;
	DI_05_ThermalBath_2DeviationAlarm AT%I*:BOOL;
	DI_05_ThermalBath_2CutOffAlarm AT%I*:BOOL;
	
	DI_06_ThermalBath_3DeviationAlarm AT%I*:BOOL;
	DI_06_ThermalBath_3CutOffAlarm AT%I*:BOOL;
	DI_06_ThermalBath_4DeviationAlarm AT%I*:BOOL;
	DI_06_ThermalBath_4CutOffAlarm AT%I*:BOOL;
	DI_06_Spare_01 AT%I*:BOOL;
	DI_06_Spare_02 AT%I*:BOOL;
	DI_06_Spare_03 AT%I*:BOOL;
	DI_06_Spare_04 AT%I*:BOOL;
	
	DO_07_SystemPowerOffLock AT%Q*:BOOL;
	DO_07_ControlCabinetLamp AT%Q*:BOOL;
	DO_07_GasCabinetLamp AT%Q*:BOOL;
	DO_07_GraphiteHeaterMC AT%Q*:BOOL;
	DO_07_ThermalBathsMC AT%Q*:BOOL;
	DO_07_VacuumPumpMC AT%Q*:BOOL;
	DO_07_LineHeatersMC AT%Q*:BOOL;
	DO_07_ResetButtonLamp AT%Q*:BOOL;
	
	DO_08_Spare_01 AT%Q*:BOOL;
	DO_08_Spare_02 AT%Q*:BOOL;
	DO_08_Spare_03 AT%Q*:BOOL;
	DO_08_Spare_04 AT%Q*:BOOL;
	DO_08_Spare_05 AT%Q*:BOOL;
	DO_08_Spare_06 AT%Q*:BOOL;
	DO_08_Spare_07 AT%Q*:BOOL;
	DO_08_Spare_08 AT%Q*:BOOL;
	
	AI_09_M01_ChalcogenRunPV AT%I*:INT;
	AI_09_M02_MORunPV AT%I*:INT;
	AI_09_M03_H2SeSupplyPV AT%I*:INT;
	AI_09_M04_H2SSupplyPV AT%I*:INT;
	
	AO_10_M01_ChalcogenRunSV AT%Q*:INT;
	AO_10_M02_MORunSV AT%Q*:INT;
	AO_10_M03_H2SeSupplySV AT%Q*:INT;
	AO_10_M04_H2SSupplySV AT%Q*:INT;
	
	AI_11_M05_Source_1TMInSupplyPV AT%I*:INT;
	AI_11_M06_Source_2TMGaSupplyPV AT%I*:INT;
	AI_11_M07_Source_3DMSeSupplyPV AT%I*:INT;
	AI_11_M08_Source_4ChalcoSupplyPV AT%I*:INT;
	
	AO_12_M05_Source_1TMInSupplySV AT%Q*:INT;
	AO_12_M06_Source_2TMGaSupplySV AT%Q*:INT;
	AO_12_M07_Source_3DMSeSupplySV AT%Q*:INT;
	AO_12_M08_Source_4ChalcoSupplySV AT%Q*:INT;
	
	AI_13_M09_LinerPurgePV AT%I*:INT;
	AI_13_M10_HeaterPurgePV AT%I*:INT;
	AI_13_M11_ChalcogenVentPV AT%I*:INT;
	AI_13_M12_MOVentPV AT%I*:INT;
	
	AO_14_M09_LinerPurgeSV AT%Q*:INT;
	AO_14_M10_HeaterPurgeSV AT%Q*:INT;
	AO_14_M11_ChalcogenVentSV AT%Q*:INT;
	AO_14_M12_MOVentSV AT%Q*:INT;
	
	AI_15_E01Source_1TMInPressurePV AT%I*:INT;
	AI_15_E02Source_2TMGaPressurePV AT%I*:INT;
	AI_15_E03Source_3DMSePressurePV AT%I*:INT;
	AI_15_E04Source_4ChalcoPressurePV AT%I*:INT;
	
	AO_16_E01Source_1TMInPressureSV AT%Q*:INT;
	AO_16_E02Source_2TMGaPressureSV AT%Q*:INT;
	AO_16_E03Source_3DMSePressureSV AT%Q*:INT;
	AO_16_E04Source_4ChalcoPressureSV AT%Q*:INT;
	
	DI_17_DP1ChalcogenDP AT%I*:INT;
	DI_17_DP2MODP AT%I*:INT;
	
	DI_18_S01N2SupplyPressPV AT%I*:INT;
	DI_18_S02H2SupplyPressPV AT%I*:INT;
	DI_18_S03H2SSupplyPressPV AT%I*:INT;
	DI_18_S04H2SeSupplyPressPV AT%I*:INT;
	
//	DI_19_LineHeaterController AT%I*:BOOL;
//	DI_20_ThermalBathx4EA AT%I*:BOOL;
	 
END_VAR

// ---- GVLs/GVL_IO_REACTOR_CABINET.TcGVL
{attribute 'qualified_only'}
VAR_GLOBAL
	DI_01_MaintenanceModeKey AT%I*:BOOL;
	DI_01_ReactorCabinetLampButton AT%I*:BOOL;
	DI_01_DORVACButton AT%I*:BOOL;
	DI_01_DORATMButton AT%I*:BOOL;
	DI_01_ReactorDoorUpButton AT%I*:BOOL;
	DI_01_ReactorDoorDownButton AT%I*:BOOL;
	DI_01_ClampLock AT%I*:BOOL;
	DI_01_ClampRelease AT%I*:BOOL;
	
	DI_02_C_WFlowSensor AT%I*:BOOL;
	DI_02_SusceptorRotationMotorFault AT%I*:BOOL;
	DI_02_VacuumPumpFail AT%I*:BOOL;
	DI_02_VacuumPumpWarning AT%I*:BOOL;
	DI_02_VacuumPumpAlarm AT%I*:BOOL;
	DI_02_VacuumPumpRunning AT%I*:BOOL;
	DI_02_VacuumPumpFBRunning AT%I*:BOOL;
	DI_02_ReactorDoorUpLimitSensor AT%I*:BOOL;
	
	DI_03_ReactorDoorDownLimitSensor AT%I*:BOOL;
	DI_03_CylinderAutoSwitch_Closed AT%I*:BOOL;
	DI_03_CylinderAutoSwitch_Opened AT%I*:BOOL;
	DI_03_ReactorCabinetDoorClose AT%I*:BOOL;
	DI_03_Spare_01 AT%I*:BOOL;
	DI_03_Spare_02 AT%I*:BOOL;
	DI_03_Spare_03 AT%I*:BOOL;
	DI_03_Spare_04 AT%I*:BOOL;
	
	DO_04_SignalTowerRed AT%Q*:BOOL;
	DO_04_SignalTowerOrange AT%Q*:BOOL;
	DO_04_SignalTowerGreen AT%Q*:BOOL;
	DO_04_SignalTowerBlue AT%Q*:BOOL;
	DO_04_SignalTowerWhite AT%Q*:BOOL;
	DO_04_SignalTowerBuzzer AT%Q*:BOOL;
	DO_04_ReactorCoverUpRelay AT%Q*:BOOL;
	DO_04_ReactorCoverDownRelay AT%Q*:BOOL;
	
	DO_05_ClampLock AT%Q*:BOOL;
	DO_05_ClampRelease AT%Q*:BOOL;
	DO_05_VacuumPumpStart_Stop AT%Q*:BOOL;
	DO_05_VacuumPumpReset AT%Q*:BOOL;
	DO_05_SusceptorRotationFWD AT%Q*:BOOL;
	DO_05_SusceptorRotationSTOP AT%Q*:BOOL;
	DO_05_SusceptorRotationAL_RST AT%Q*:BOOL;
	DO_05_DORVACButtonLamp AT%Q*:BOOL;
	
	DO_06_DORATMButtonLamp AT%Q*:BOOL;
	DO_06_ReactorCoverUpButtonLamp AT%Q*:BOOL;
	DO_06_ReactorCoverDownButtonLamp AT%Q*:BOOL;
	DO_06_ClampLockButtonLamp AT%Q*:BOOL;
	DO_06_ClampReleaseButtonLamp AT%Q*:BOOL;
	DO_06_ReactorCabinetLamp AT%Q*:BOOL;
	DO_06_Spare07 AT%Q*:BOOL;
	DO_06_Spare08 AT%Q*:BOOL;
	
	AI_07_P02_ReactorPressure10TorrPV AT%I*:INT;
	AI_07_P03_ExhaustPressurePV AT%I*:INT;
	AI_07_S05_DORPressurePV AT%I*:INT;
	AI_07_Spare_04 AT%I*:INT;

	AI_08_R01SusceptorRotationPV AT%I*:INT;
	AI_08_Spare_02 AT%I*:INT;
	AI_08_Spare_03 AT%I*:INT;
	AI_08_Spare_04 AT%I*:INT;
	
	AO_09_P03_ExhaustPressureAM215Input AT%Q*:INT;
	AO_09_R01_SusceptorRotationSV AT%Q*:INT;
	AO_09_Spare_03 AT%Q*:INT;
	AO_09_Spare_04 AT%Q*:INT;
	
	AI_10_R04S_HCoolingWaterPV AT%I*:INT;
	AI_10_Spare_02 AT%I*:INT;
	AI_10_Spare_03 AT%I*:INT;
	AI_10_Spare_04 AT%I*:INT;

 
END_VAR

// ---- GVLs/GVL_Serial.TcGVL
{attribute 'qualified_only'}
VAR_GLOBAL
	TxBufferTB : ComBuffer; (* Receive data buffer; used with all receive function blocks *)
	RxBufferTB : ComBuffer; (* Transmit data buffer; used with all receive function blocks *)
	
	stIn_KL6031_TB AT %I*	: KL6inData22B;	(* linked to the KL6001 in the TwinCAT System Manager *)
	stOut_KL6031_TB AT %Q*	: KL6outData22B;	(* linked to the KL6001 in the TwinCAT System Manager *)	
	
	LineHeater_data_1	:ST_LineHeater_Data;
	LineHeater_data_2	:ST_LineHeater_Data;
	
	(*HORIBA MFC용 *)
	fbSL : SerialLineControl;
	
	
	TxBufferTB_MFC : ComBuffer; (* Receive data buffer; used with all receive function blocks *)
	RxBufferTB_MFC : ComBuffer; (* Transmit data buffer; used with all receive function blocks *)
	
	EL6021_In AT %I* : ARRAY[0..21] OF BYTE; (* Terminal → PLC *)
	EL6021_Out AT %Q* : ARRAY[0..21] OF BYTE; (* PLC → Terminal *)
	
END_VAR

// ---- POUs/MAIN.TcPOU
PROGRAM MAIN
VAR
	controlMode	: E_ControlMode := E_ControlMode.Manual;
	prevControlMode : E_ControlMode := controlMode;
END_VAR

F_Variable_Valve();
F_Variable_DeviceLink();
F_Variable_FromUI();
F_Variable_FromUI_Interlock();
F_Variable_TODevice();
F_Variable_ToUI_InputState();
GVL.fbLineHeater_Manager(RData_Module_1=>GVL_Serial.LineHeater_data_1,RData_Module_2=>GVL_Serial.LineHeater_data_2);


P11_E3508(); //Temp Controller
P12_IQ_PLUS(); //Throttle Valve Controller
P13_LineHeater();
P14_ThermalBath();
P15_RotationOperation();
P16_CoverOperation();
P17_DOROperation();
P22_Background_ThermalBath();


IF controlMode <> E_ControlMode.Priority THEN
	IF controlMode <> GVL_INTERFACE_UI.mainPRGControl.controlModeCmd THEN
		IF GVL_INTERFACE_UI.mainPRGControl.controlModeCmd = E_ControlMode.Priority THEN
			prevControlMode := controlMode;
		END_IF
		GVL_INTERFACE_UI.mainPRGControl.controlMode := controlMode := GVL_INTERFACE_UI.mainPRGControl.controlModeCmd;
	END_IF
END_IF

CASE controlMode OF
	E_ControlMode.Manual:
		P30_ManualControl();
	
	E_ControlMode.Recipe:
		P50_RecipeControl(); //레시피 콘트론
		
	E_ControlMode.Priority:
		P31_PriorityControl();
		IF P31_PriorityControl.complete = TRUE THEN
			GVL_INTERFACE_UI.mainPRGControl.controlMode := controlMode := prevControlMode;
			GVL_INTERFACE_UI.mainPRGControl.controlModeCmd := controlMode;
		END_IF
END_CASE

P60_UpdatePV();
P70_Interface();
P90_Interlock();
P91_Monitoring();
P92_Maintenance();

END_PROGRAM

// ---- POUs/VARIABLE_LINK/F_Variable_Valve.TcPOU
FUNCTION F_Variable_Valve: BOOL

GVL_IO_VALVE.DO_00_V01ChalcogenCarrierChange :=GVL_INTERFACE_UI.aOutputSolValve[1];
GVL_IO_VALVE.DO_00_V02MOCarreirChange :=GVL_INTERFACE_UI.aOutputSolValve[2];
GVL_IO_VALVE.DO_00_V03H2SeSourceChange:=GVL_INTERFACE_UI.aOutputSolValve[3];
GVL_IO_VALVE.DO_00_V04H2SSourceChange :=GVL_INTERFACE_UI.aOutputSolValve[4];
GVL_IO_VALVE.DO_00_V05Source_1TMInCarrierChange :=GVL_INTERFACE_UI.aOutputSolValve[5];
GVL_IO_VALVE.DO_00_V06Source_1TMInBypass :=GVL_INTERFACE_UI.aOutputSolValve[6];
GVL_IO_VALVE.DO_00_V07Source_2TMGaCarrierChange :=GVL_INTERFACE_UI.aOutputSolValve[7];
GVL_IO_VALVE.DO_00_V08Source_2TMGaBypass :=GVL_INTERFACE_UI.aOutputSolValve[8];
GVL_IO_VALVE.DO_00_V09Source_3DMSeCarrierChange :=GVL_INTERFACE_UI.aOutputSolValve[9];
GVL_IO_VALVE.DO_00_V10Source_3DMSeBypass :=GVL_INTERFACE_UI.aOutputSolValve[10];
GVL_IO_VALVE.DO_00_V11Source_4ChalcogenCarrierChange :=GVL_INTERFACE_UI.aOutputSolValve[11];
GVL_IO_VALVE.DO_00_V12Source_4ChalcogenBypass :=GVL_INTERFACE_UI.aOutputSolValve[12];
GVL_IO_VALVE.DO_00_V13ReactorPurgeCarrierChange :=GVL_INTERFACE_UI.aOutputSolValve[13];
GVL_IO_VALVE.DO_00_V14Source_1TMInManifoldRun :=GVL_INTERFACE_UI.aOutputSolValve[14];
GVL_IO_VALVE.DO_00_V15Source_2TMGaManifoldRun :=GVL_INTERFACE_UI.aOutputSolValve[15];
GVL_IO_VALVE.DO_00_V16Source_3DMSeManifoldRun :=GVL_INTERFACE_UI.aOutputSolValve[16];
GVL_IO_VALVE.DO_00_V17GasH2SeManifoldRun :=GVL_INTERFACE_UI.aOutputSolValve[17];
GVL_IO_VALVE.DO_00_V18GasH2SManifoldRun  :=GVL_INTERFACE_UI.aOutputSolValve[18];
GVL_IO_VALVE.DO_00_V19Source_4ChalcogenManifoldRun :=GVL_INTERFACE_UI.aOutputSolValve[19];
GVL_IO_VALVE.DO_00_V20VentPress_Change :=GVL_INTERFACE_UI.aOutputSolValve[20];
GVL_IO_VALVE.DO_00_V21PumpByPass :=NOT GVL_INTERFACE_UI.aOutputSolValve[21];
GVL_IO_VALVE.DO_00_V22DORVaccumON :=GVL_INTERFACE_UI.aOutputSolValve[22];
GVL_IO_VALVE.DO_00_V23DORFilling  :=GVL_INTERFACE_UI.aOutputSolValve[23];
GVL_IO_VALVE.DO_00_V24Source_1LeakTest_IN :=GVL_INTERFACE_UI.aOutputSolValve[24];
GVL_IO_VALVE.DO_00_V25Source_1LeakTest_OUT:=GVL_INTERFACE_UI.aOutputSolValve[25];
GVL_IO_VALVE.DO_00_V26Source_2LeakTest_IN :=GVL_INTERFACE_UI.aOutputSolValve[26];
GVL_IO_VALVE.DO_00_V27Source_2LeakTest_OUT:=GVL_INTERFACE_UI.aOutputSolValve[27];
GVL_IO_VALVE.DO_00_V28Source_3LeakTest_IN :=GVL_INTERFACE_UI.aOutputSolValve[28];
GVL_IO_VALVE.DO_00_V29Source_3LeakTest_OUT:=GVL_INTERFACE_UI.aOutputSolValve[29];
GVL_IO_VALVE.DO_00_V30Source_4LeakTest_IN :=GVL_INTERFACE_UI.aOutputSolValve[30];
GVL_IO_VALVE.DO_00_V31Source_4LeakTest_OUT:=GVL_INTERFACE_UI.aOutputSolValve[31];
GVL_IO_VALVE.DO_00_V32SourceVacuumON :=GVL_INTERFACE_UI.aOutputSolValve[32];

END_FUNCTION

// ---- POUs/VARIABLE_LINK/F_Variable_DeviceLink.TcPOU
FUNCTION F_Variable_DeviceLink: BOOL



//GVL_IO.io.digital.aDigitalInputIO[1]:=GVL_IO_GAS_CABINET.DI_01_ResetButton ;
//GVL_IO.io.digital.aDigitalInputIO[2]:=GVL_IO_GAS_CABINET.DI_01_GasCabinetLampButton ;//ok
//GVL_IO.io.digital.aDigitalInputIO[3]:=GVL_IO_GAS_CABINET.DI_01_PneumaticPressureSensor ;
//GVL_IO.io.digital.aDigitalInputIO[4]:=GVL_IO_GAS_CABINET.DI_01_GasCabinetDoorClose ;
//GVL_IO.io.digital.aDigitalInputIO[5]:=GVL_IO_GAS_CABINET.DI_01_ControlCabinetDoorClose ;
//GVL_IO.io.digital.aDigitalInputIO[6]:=GVL_IO_GAS_CABINET.DI_01_SMPS_1Alarm ;
//GVL_IO.io.digital.aDigitalInputIO[7]:=GVL_IO_GAS_CABINET.DI_01_SMPS_2Alarm ;
//GVL_IO.io.digital.aDigitalInputIO[8]:=GVL_IO_GAS_CABINET.DI_01_SMPS_3Alarm ;

//GVL_IO.io.digital.aDigitalInputIO[9]:=GVL_IO_GAS_CABINET.DI_02_SMPS_4Alarm ;
//GVL_IO.io.digital.aDigitalInputIO[10]:=GVL_IO_GAS_CABINET.DI_02_GraphiteHeaterELCB ;
//GVL_IO.io.digital.aDigitalInputIO[11]:=GVL_IO_GAS_CABINET.DI_02_ThermalBathsELCB ;
//GVL_IO.io.digital.aDigitalInputIO[12]:=GVL_IO_GAS_CABINET.DI_02_VacuumPumpELCB ;
//GVL_IO.io.digital.aDigitalInputIO[13]:=GVL_IO_GAS_CABINET.DI_02_LineHeatersELCB ;
//GVL_IO.io.digital.aDigitalInputIO[14]:=GVL_IO_GAS_CABINET.DI_02_RotationMotorCP ;
//GVL_IO.io.digital.aDigitalInputIO[15]:=GVL_IO_GAS_CABINET.DI_02_CoverLiftMotorCP ;
//GVL_IO.io.digital.aDigitalInputIO[16]:=GVL_IO_GAS_CABINET.DI_02_T_VCP ;

//GVL_IO.io.digital.aDigitalInputIO[17]:=GVL_IO_GAS_CABINET.DI_03_GasDetectorCP ;
//GVL_IO.io.digital.aDigitalInputIO[18]:=GVL_IO_GAS_CABINET.DI_03_CabinetLampsCP ;
//GVL_IO.io.digital.aDigitalInputIO[19]:=GVL_IO_GAS_CABINET.DI_03_MFCPowerCP ;
//GVL_IO.io.digital.aDigitalInputIO[20]:=GVL_IO_GAS_CABINET.DI_03_LineHeater_1CP ;
//GVL_IO.io.digital.aDigitalInputIO[21]:=GVL_IO_GAS_CABINET.DI_03_LineHeater_2CP ;
//GVL_IO.io.digital.aDigitalInputIO[22]:=GVL_IO_GAS_CABINET.DI_03_LineHeater_3CP ;
//GVL_IO.io.digital.aDigitalInputIO[23]:=GVL_IO_GAS_CABINET.DI_03_LineHeater_4CP ;
//GVL_IO.io.digital.aDigitalInputIO[24]:=GVL_IO_GAS_CABINET.DI_03_LineHeater_5CP ;

//GVL_IO.io.digital.aDigitalInputIO[25]:=GVL_IO_GAS_CABINET.DI_04_LineHeater_6CP ;
//GVL_IO.io.digital.aDigitalInputIO[26]:=GVL_IO_GAS_CABINET.DI_04_LineHeater_7CP ;
//GVL_IO.io.digital.aDigitalInputIO[27]:=GVL_IO_GAS_CABINET.DI_04_LineHeater_8CP ;
//GVL_IO.io.digital.aDigitalInputIO[28]:=GVL_IO_GAS_CABINET.DI_04_GasDetectorH2 ;
//GVL_IO.io.digital.aDigitalInputIO[29]:=GVL_IO_GAS_CABINET.DI_04_GasDetectorH2S ;
//GVL_IO.io.digital.aDigitalInputIO[30]:=GVL_IO_GAS_CABINET.DI_04_GasDetectorH2Se ;
//GVL_IO.io.digital.aDigitalInputIO[31]:=GVL_IO_GAS_CABINET.DI_04_FireSensor ;
//GVL_IO.io.digital.aDigitalInputIO[32]:=GVL_IO_GAS_CABINET.DI_04_ExternalScrubberFault ;

//GVL_IO.io.digital.aDigitalInputIO[33]:=GVL_IO_GAS_CABINET.DI_05_ExternalH2GasCabinetFault ;
//GVL_IO.io.digital.aDigitalInputIO[34]:=GVL_IO_GAS_CABINET.DI_05_ExternalH2SGasCabinetFault ;
//GVL_IO.io.digital.aDigitalInputIO[35]:=GVL_IO_GAS_CABINET.DI_05_ExternalH2SeGasCabinetFault ;
//GVL_IO.io.digital.aDigitalInputIO[36]:=GVL_IO_GAS_CABINET.DI_05_ExternalUserInputAlarm ;
//GVL_IO.io.digital.aDigitalInputIO[37]:=GVL_IO_GAS_CABINET.DI_05_ThermalBath_1DeviationAlarm ;
//GVL_IO.io.digital.aDigitalInputIO[38]:=GVL_IO_GAS_CABINET.DI_05_ThermalBath_1CutOffAlarm ;
//GVL_IO.io.digital.aDigitalInputIO[39]:=GVL_IO_GAS_CABINET.DI_05_ThermalBath_2DeviationAlarm ;
//GVL_IO.io.digital.aDigitalInputIO[40]:=GVL_IO_GAS_CABINET.DI_05_ThermalBath_2CutOffAlarm ;

//GVL_IO.io.digital.aDigitalInputIO[41]:=GVL_IO_GAS_CABINET.DI_06_ThermalBath_3DeviationAlarm ;
//GVL_IO.io.digital.aDigitalInputIO[41]:=GVL_IO_GAS_CABINET.DI_06_ThermalBath_3CutOffAlarm ;
//GVL_IO.io.digital.aDigitalInputIO[42]:=GVL_IO_GAS_CABINET.DI_06_ThermalBath_4DeviationAlarm ;
//GVL_IO.io.digital.aDigitalInputIO[43]:=GVL_IO_GAS_CABINET.DI_06_ThermalBath_4CutOffAlarm ;
//GVL_IO.io.digital.aDigitalInputIO[44]:=GVL_IO_GAS_CABINET.DI_06_Spare_01 ;
//GVL_IO.io.digital.aDigitalInputIO[45]:=GVL_IO_GAS_CABINET.DI_06_Spare_02 ;
//GVL_IO.io.digital.aDigitalInputIO[46]:=GVL_IO_GAS_CABINET.DI_06_Spare_03 ;
//GVL_IO.io.digital.aDigitalInputIO[47]:=GVL_IO_GAS_CABINET.DI_06_Spare_04 ;

//GVL_IO.io.digital.aDigitalInputIO[48]:=GVL_IO_REACTOR_CABINET.DI_01_MaintenanceModeKey ;
//GVL_IO.io.digital.aDigitalInputIO[49]:=GVL_IO_REACTOR_CABINET.DI_01_ReactorCabinetLampButton ;
//GVL_IO.io.digital.aDigitalInputIO[50]:=GVL_IO_REACTOR_CABINET.DI_01_DORVACButton ; //Sheet에서는 빠짐
//GVL_IO.io.digital.aDigitalInputIO[51]:=GVL_IO_REACTOR_CABINET.DI_01_DORATMButton ;//Sheet에서는 빠짐
//GVL_IO.io.digital.aDigitalInputIO[52]:=GVL_IO_REACTOR_CABINET.DI_01_ReactorDoorUpButton ;//Sheet에서는 빠짐
//GVL_IO.io.digital.aDigitalInputIO[53]:=GVL_IO_REACTOR_CABINET.DI_01_ReactorDoorDownButton ;//Sheet에서는 빠짐
//GVL_IO.io.digital.aDigitalInputIO[54]:=GVL_IO_REACTOR_CABINET.DI_01_ClampLock ;//Sheet에서는 빠짐
//GVL_IO.io.digital.aDigitalInputIO[55]:=GVL_IO_REACTOR_CABINET.DI_01_ClampRelease ;//Sheet에서는 빠짐

//GVL_IO.io.digital.aDigitalInputIO[56]:=GVL_IO_REACTOR_CABINET.DI_02_C_WFlowSensor ;
//GVL_IO.io.digital.aDigitalInputIO[57]:=GVL_IO_REACTOR_CABINET.DI_02_SusceptorRotationMotorFault ;
//GVL_IO.io.digital.aDigitalInputIO[58]:=GVL_IO_REACTOR_CABINET.DI_02_VacuumPumpFail ;
//GVL_IO.io.digital.aDigitalInputIO[59]:=GVL_IO_REACTOR_CABINET.DI_02_VacuumPumpWarning ;
//GVL_IO.io.digital.aDigitalInputIO[60]:=GVL_IO_REACTOR_CABINET.DI_02_VacuumPumpAlarm ;
//GVL_IO.io.digital.aDigitalInputIO[61]:=GVL_IO_REACTOR_CABINET.DI_02_VacuumPumpFBRunning ;
//GVL_IO.io.digital.aDigitalInputIO[62]:=GVL_IO_REACTOR_CABINET.DI_02_VacuumPumpFBRunning ;
//GVL_IO.io.digital.aDigitalInputIO[63]:=GVL_IO_REACTOR_CABINET.DI_02_ReactorDoorUpLimitSensor ;

//GVL_IO.io.digital.aDigitalInputIO[64]:=GVL_IO_REACTOR_CABINET.DI_03_ReactorDoorDownLimitSensor ;
//GVL_IO.io.digital.aDigitalInputIO[65]:=GVL_IO_REACTOR_CABINET.DI_03_CylinderAutoSwitch_Closed ;
//GVL_IO.io.digital.aDigitalInputIO[66]:=GVL_IO_REACTOR_CABINET.DI_03_CylinderAutoSwitch_Opened ;
//GVL_IO.io.digital.aDigitalInputIO[67]:=GVL_IO_REACTOR_CABINET.DI_03_ReactorCabinetDoorClose ;
//GVL_IO.io.digital.aDigitalInputIO[68]:=GVL_IO_REACTOR_CABINET.DI_03_Spare_01 ;
//GVL_IO.io.digital.aDigitalInputIO[69]:=GVL_IO_REACTOR_CABINET.DI_03_Spare_02 ;
//GVL_IO.io.digital.aDigitalInputIO[70]:=GVL_IO_REACTOR_CABINET.DI_03_Spare_03 ;
//GVL_IO.io.digital.aDigitalInputIO[71]:=GVL_IO_REACTOR_CABINET.DI_03_Spare_04 ;


//GVL_IO.io.digital.aDigitalOutputIO[1]:=GVL_IO_GAS_CABINET.DO_07_SystemPowerOffLock ; //Sheet에서는 빠짐
//GVL_IO.io.digital.aDigitalOutputIO[2]:=GVL_IO_GAS_CABINET.DO_07_ControlCabinetLamp ;//Sheet에서는 빠짐
//GVL_IO.io.digital.aDigitalOutputIO[3]:=GVL_IO_GAS_CABINET.DO_07_GasCabinetLamp ;//Sheet에서는 빠짐
//GVL_IO.io.digital.aDigitalOutputIO[4]:=GVL_IO_GAS_CABINET.DO_07_GraphiteHeaterMC ;//Sheet에서는 빠짐
//GVL_IO.io.digital.aDigitalOutputIO[5]:=GVL_IO_GAS_CABINET.DO_07_ThermalBathsMC ;//Sheet에서는 빠짐
//GVL_IO.io.digital.aDigitalOutputIO[6]:=GVL_IO_GAS_CABINET.DO_07_VacuumPumpMC ;//Sheet에서는 빠짐
//GVL_IO.io.digital.aDigitalOutputIO[7]:=GVL_IO_GAS_CABINET.DO_07_LineHeatersMC ;//Sheet에서는 빠짐
//GVL_IO.io.digital.aDigitalOutputIO[8]:=GVL_IO_GAS_CABINET.DO_07_ResetButtonLamp ;//Sheet에서는 빠짐

//GVL_IO.io.digital.aDigitalOutputIO[9]:=GVL_IO_GAS_CABINET.DO_08_Spare_01 ;
//GVL_IO.io.digital.aDigitalOutputIO[10]:=GVL_IO_GAS_CABINET.DO_08_Spare_02 ;
//GVL_IO.io.digital.aDigitalOutputIO[11]:=GVL_IO_GAS_CABINET.DO_08_Spare_03 ;
//GVL_IO.io.digital.aDigitalOutputIO[12]:=GVL_IO_GAS_CABINET.DO_08_Spare_04 ;
//GVL_IO.io.digital.aDigitalOutputIO[13]:=GVL_IO_GAS_CABINET.DO_08_Spare_05 ;
//GVL_IO.io.digital.aDigitalOutputIO[14]:=GVL_IO_GAS_CABINET.DO_08_Spare_06 ;
//GVL_IO.io.digital.aDigitalOutputIO[15]:=GVL_IO_GAS_CABINET.DO_08_Spare_07 ;
//GVL_IO.io.digital.aDigitalOutputIO[16]:=GVL_IO_GAS_CABINET.DO_08_Spare_08 ;

//GVL_IO.io.digital.aDigitalOutputIO[17]:=GVL_IO_REACTOR_CABINET.DO_04_SignalTowerRed ;
//GVL_IO.io.digital.aDigitalOutputIO[18]:=GVL_IO_REACTOR_CABINET.DO_04_SignalTowerOrange ;
//GVL_IO.io.digital.aDigitalOutputIO[19]:=GVL_IO_REACTOR_CABINET.DO_04_SignalTowerGreen ;
//GVL_IO.io.digital.aDigitalOutputIO[20]:=GVL_IO_REACTOR_CABINET.DO_04_SignalTowerBlue ;
//GVL_IO.io.digital.aDigitalOutputIO[21]:=GVL_IO_REACTOR_CABINET.DO_04_SignalTowerWhite ;
//GVL_IO.io.digital.aDigitalOutputIO[22]:=GVL_IO_REACTOR_CABINET.DO_04_SignalTowerBuzzer ;
//GVL_IO.io.digital.aDigitalOutputIO[23]:=GVL_IO_REACTOR_CABINET.DO_04_ReactorCoverUpRelay ; //Sheet에서는 빠짐
//GVL_IO.io.digital.aDigitalOutputIO[24]:=GVL_IO_REACTOR_CABINET.DO_04_ReactorCoverDownRelay ;//Sheet에서는 빠짐

//GVL_IO.io.digital.aDigitalOutputIO[25]:=GVL_IO_REACTOR_CABINET.DO_05_ClampLock ;
//GVL_IO.io.digital.aDigitalOutputIO[26]:=GVL_IO_REACTOR_CABINET.DO_05_ClampRelease ;
//GVL_IO.io.digital.aDigitalOutputIO[27]:=GVL_IO_REACTOR_CABINET.DO_05_VacuumPumpStart_Stop ;//Sheet에서는 빠짐
//GVL_IO.io.digital.aDigitalOutputIO[28]:=GVL_IO_REACTOR_CABINET.DO_05_VacuumPumpReset ;//Sheet에서는 빠짐
//GVL_IO.io.digital.aDigitalOutputIO[29]:=GVL_IO_REACTOR_CABINET.DO_05_SusceptorRotationFWD ;
//GVL_IO.io.digital.aDigitalOutputIO[30]:=GVL_IO_REACTOR_CABINET.DO_05_SusceptorRotationSTOP ;
//GVL_IO.io.digital.aDigitalOutputIO[31]:=GVL_IO_REACTOR_CABINET.DO_05_SusceptorRotationAL_RST ;//Sheet에서는 빠짐
//GVL_IO.io.digital.aDigitalOutputIO[32]:=GVL_IO_REACTOR_CABINET.DO_05_DORVACButtonLamp ;//Sheet에서는 빠짐

//GVL_IO.io.digital.aDigitalOutputIO[33]:=GVL_IO_REACTOR_CABINET.DO_06_DORATMButtonLamp ;//Sheet에서는 빠짐
//GVL_IO.io.digital.aDigitalOutputIO[34]:=GVL_IO_REACTOR_CABINET.DO_06_ReactorCoverUpButtonLamp ;//Sheet에서는 빠짐
//GVL_IO.io.digital.aDigitalOutputIO[35]:=GVL_IO_REACTOR_CABINET.DO_06_ReactorCoverDownButtonLamp ;//Sheet에서는 빠짐
//GVL_IO.io.digital.aDigitalOutputIO[36]:=GVL_IO_REACTOR_CABINET.DO_06_ClampLockButtonLamp ;//Sheet에서는 빠짐
//GVL_IO.io.digital.aDigitalOutputIO[37]:=GVL_IO_REACTOR_CABINET.DO_06_ClampReleaseButtonLamp ;//Sheet에서는 빠짐
//GVL_IO.io.digital.aDigitalOutputIO[38]:=GVL_IO_REACTOR_CABINET.DO_06_ReactorCabinetLamp ;//Sheet에서는 빠짐
//GVL_IO.io.digital.aDigitalOutputIO[39]:=GVL_IO_REACTOR_CABINET.DO_06_Spare07 ;//Sheet에서는 빠짐
//GVL_IO.io.digital.aDigitalOutputIO[40]:=GVL_IO_REACTOR_CABINET.DO_06_Spare08 ;//Sheet에서는 빠짐


//GVL_IO.io.analog.aAnalogInputIO[1]:=GVL_IO_GAS_CABINET.AI_09_M01_ChalcogenRunPV ;
//GVL_IO.io.analog.aAnalogInputIO[2]:=GVL_IO_GAS_CABINET.AI_09_M02_MORunPV ;
//GVL_IO.io.analog.aAnalogInputIO[3]:=GVL_IO_GAS_CABINET.AI_09_M03_H2SeSupplyPV ;
//GVL_IO.io.analog.aAnalogInputIO[4]:=GVL_IO_GAS_CABINET.AI_09_M04_H2SSupplyPV ;
//GVL_IO.io.analog.aAnalogInputIO[5]:=GVL_IO_GAS_CABINET.AI_11_M05_Source_1TMInSupplyPV ;
//GVL_IO.io.analog.aAnalogInputIO[6]:=GVL_IO_GAS_CABINET.AI_11_M06_Source_2TMGaSupplyPV ;
//GVL_IO.io.analog.aAnalogInputIO[7]:=GVL_IO_GAS_CABINET.AI_11_M07_Source_3DMSeSupplyPV ;
//GVL_IO.io.analog.aAnalogInputIO[8]:=GVL_IO_GAS_CABINET.AI_11_M08_Source_4ChalcoSupplyPV ;
//GVL_IO.io.analog.aAnalogInputIO[9]:=GVL_IO_GAS_CABINET.AI_13_M09_LinerPurgePV ;
//GVL_IO.io.analog.aAnalogInputIO[10]:=GVL_IO_GAS_CABINET.AI_13_M10_HeaterPurgePV ;
//GVL_IO.io.analog.aAnalogInputIO[11]:=GVL_IO_GAS_CABINET.AI_13_M11_ChalcogenVentPV ;
//GVL_IO.io.analog.aAnalogInputIO[12]:=GVL_IO_GAS_CABINET.AI_13_M12_MOVentPV ;
//GVL_IO.io.analog.aAnalogInputIO[13]:=GVL_IO_GAS_CABINET.AI_15_E01Source_1TMInPressurePV ;
//GVL_IO.io.analog.aAnalogInputIO[14]:=GVL_IO_GAS_CABINET.AI_15_E02Source_2TMGaPressurePV ;
//GVL_IO.io.analog.aAnalogInputIO[15]:=GVL_IO_GAS_CABINET.AI_15_E03Source_3DMSePressurePV ;
//GVL_IO.io.analog.aAnalogInputIO[16]:=GVL_IO_GAS_CABINET.AI_15_E04Source_4ChalcoPressurePV ;


//GVL_IO.io.analog.aAnalogInputIO[17]:=GVL_IO_REACTOR_CABINET.AI_08_R01SusceptorRotationPV ;
//GVL_IO.io.analog.aAnalogInputIO[18]:=GVL_IO_REACTOR_CABINET.AI_07_P02_ReactorPressure10TorrPV;
//GVL_IO.io.analog.aAnalogInputIO[19]:=GVL_IO_REACTOR_CABINET.AI_07_P03_ExhaustPressurePV ;
//GVL_IO.io.analog.aAnalogInputIO[20]:=GVL_IO_REACTOR_CABINET.AI_07_S05_DORPressurePV ;

//GVL_IO.io.analog.aAnalogInputIO[21]:=GVL_IO_GAS_CABINET.DI_18_S01N2SupplyPressPV ;
//GVL_IO.io.analog.aAnalogInputIO[22]:=GVL_IO_GAS_CABINET.DI_18_S02H2SupplyPressPV ;
//GVL_IO.io.analog.aAnalogInputIO[23]:=GVL_IO_GAS_CABINET.DI_18_S03H2SSupplyPressPV ;
//GVL_IO.io.analog.aAnalogInputIO[24]:=GVL_IO_GAS_CABINET.DI_18_S04H2SeSupplyPressPV ;
//GVL_IO.io.analog.aAnalogInputIO[25]:=GVL_IO_REACTOR_CABINET.AI_10_R04S_HCoolingWaterPV ;


//GVL_IO.io.analog.aAnalogInputIO[26]:=GVL_IO_GAS_CABINET.DI_17_DP1ChalcogenDP ;
//GVL_IO.io.analog.aAnalogInputIO[27]:=GVL_IO_GAS_CABINET.DI_17_DP2MODP ;


////GVL_IO.aAnalogInputIO[24]:=GVL_IO_REACTOR_CABINET.AI_07_Spare_04 ;
////GVL_IO.aAnalogInputIO[26]:=GVL_IO_REACTOR_CABINET.AI_08_Spare_02 ;
////GVL_IO.aAnalogInputIO[27]:=GVL_IO_REACTOR_CABINET.AI_08_Spare_03 ;
////GVL_IO.aAnalogInputIO[28]:=GVL_IO_REACTOR_CABINET.AI_08_Spare_04 ;


////GVL_IO.aAnalogInputIO[30]:=GVL_IO_REACTOR_CABINET.AI_10_Spare_02 ;
////GVL_IO.aAnalogInputIO[31]:=GVL_IO_REACTOR_CABINET.AI_10_Spare_03 ;
////GVL_IO.aAnalogInputIO[32]:=GVL_IO_REACTOR_CABINET.AI_10_Spare_04 ;


//GVL_IO_GAS_CABINET.AO_10_M01_ChalcogenRunSV :=GVL_IO.IO.analog.aAnalogOutputIO[1];
//GVL_IO_GAS_CABINET.AO_10_M02_MORunSV:=GVL_IO.IO.analog.aAnalogOutputIO[2];
//GVL_IO_GAS_CABINET.AO_10_M03_H2SeSupplySV:=GVL_IO.IO.analog.aAnalogOutputIO[3];
//GVL_IO_GAS_CABINET.AO_10_M04_H2SSupplySV :=GVL_IO.IO.analog.aAnalogOutputIO[4];

//GVL_IO_GAS_CABINET.AO_12_M05_Source_1TMInSupplySV :=GVL_IO.IO.analog.aAnalogOutputIO[5];
//GVL_IO_GAS_CABINET.AO_12_M06_Source_2TMGaSupplySV :=GVL_IO.IO.analog.aAnalogOutputIO[6];
//GVL_IO_GAS_CABINET.AO_12_M07_Source_3DMSeSupplySV :=GVL_IO.IO.analog.aAnalogOutputIO[7];
//GVL_IO_GAS_CABINET.AO_12_M08_Source_4ChalcoSupplySV :=GVL_IO.IO.analog.aAnalogOutputIO[8];
//GVL_IO_GAS_CABINET.AO_14_M09_LinerPurgeSV :=GVL_IO.IO.analog.aAnalogOutputIO[9];
//GVL_IO_GAS_CABINET.AO_14_M10_HeaterPurgeSV :=GVL_IO.IO.analog.aAnalogOutputIO[10];
//GVL_IO_GAS_CABINET.AO_14_M11_ChalcogenVentSV :=GVL_IO.IO.analog.aAnalogOutputIO[11];
//GVL_IO_GAS_CABINET.AO_14_M12_MOVentSV :=GVL_IO.IO.analog.aAnalogOutputIO[12];
//GVL_IO_GAS_CABINET.AO_16_E01Source_1TMInPressureSV :=GVL_IO.IO.analog.aAnalogOutputIO[13];
//GVL_IO_GAS_CABINET.AO_16_E02Source_2TMGaPressureSV :=GVL_IO.IO.analog.aAnalogOutputIO[14];
//GVL_IO_GAS_CABINET.AO_16_E03Source_3DMSePressureSV :=GVL_IO.IO.analog.aAnalogOutputIO[15];
//GVL_IO_GAS_CABINET.AO_16_E04Source_4ChalcoPressureSV :=GVL_IO.IO.analog.aAnalogOutputIO[16];

////GVL_IO_REACTOR_CABINET.AO_09_P03_ExhaustPressureAM215Input:=GVL_IO.IO.analog.aAnalogOutputIO[17];

//GVL_IO_REACTOR_CABINET.AO_09_P03_ExhaustPressureAM215Input:=GVL_IO_REACTOR_CABINET.AI_07_P03_ExhaustPressurePV;


//GVL_IO_REACTOR_CABINET.AO_09_R01_SusceptorRotationSV:=GVL_IO.IO.analog.aAnalogOutputIO[18];
//GVL_IO_REACTOR_CABINET.AO_09_Spare_03:=GVL_IO.IO.analog.aAnalogOutputIO[19];
//GVL_IO_REACTOR_CABINET.AO_09_Spare_04 :=GVL_IO.IO.analog.aAnalogOutputIO[20];

END_FUNCTION

// ---- POUs/VARIABLE_LINK/F_Variable_FromUI.TcPOU
FUNCTION F_Variable_FromUI: BOOL


VAR
	rRotationAlarm_Reset: R_TRIG;
	
	Rotation_Shift: WORD;
END_VAR

//jhkang_251112
//////UI에서 Write하는 Command
////아래 MC는 Maint 모드에서만 조작 가능
////GVL_COMMAND_FROM_UI.CMD_HEATER_MAIN_MC_ON:= GVL_IO.aOutputCmd[1].0;
////GVL_COMMAND_FROM_UI.CMD_THERMAL_BACH_MC_ON:= GVL_IO.aOutputCmd[1].1;
////GVL_COMMAND_FROM_UI.CMD_VACUUM_PUMP_MC_ON:= GVL_IO.aOutputCmd[1].2;
////GVL_COMMAND_FROM_UI.CMD_LINE_HEATER_MC_ON := GVL_IO.aOutputCmd[1].3;

//GVL_COMMAND_FROM_UI.CMD_VACUUM_PUMP_ON := GVL_IO.aOutputCmd[1];
//GVL_COMMAND_FROM_UI.CMD_VACUUM_PUMP_RESET:= GVL_IO.aOutputCmd[1].7;

//GVL_COMMAND_FROM_UI.CMD_ROTATION_START:= GVL_IO.aOutputCmd[1].8;
//GVL_COMMAND_FROM_UI.CMD_ROTATION_RESET := GVL_IO.aOutputCmd[1].10;

////jhkang 하드웨어로 구성 되어 있어야 하는데 아직 구성 안됨 := GVL_IO.aOutputCmd[1].10;
//GVL_COMMAND_FROM_UI.CMD_E3508_MAN_AUTO := GVL_IO.aOutputCmd[1].12;(*True:Manual  False:auto*)
//GVL_COMMAND_FROM_UI.CMD_THROTTLE_PRESSURE_POSITION_MODE := GVL_IO.aOutputCmd[1].13;//true: Pressure False:Position

//GVL_COMMAND_FROM_UI.CMD_THROTTLE_OUTPUT_MODE:= WORD_TO_USINT(GVL_IO.aOutputCmd[2]); //Throttle Valve Mode Setting 0:Normal 1:Close 2:Open 3:Hold 4:Reset

//GVL_IO_GAS_CABINET.DO_07_GraphiteHeaterMC :=  GVL_COMMAND_FROM_UI.CMD_HEATER_MAIN_MC_ON;
//GVL_IO_GAS_CABINET.DO_07_ThermalBathsMC :=  GVL_COMMAND_FROM_UI.CMD_THERMAL_BACH_MC_ON;
//GVL_IO_GAS_CABINET.DO_07_VacuumPumpMC :=  GVL_COMMAND_FROM_UI.CMD_VACUUM_PUMP_MC_ON;
//GVL_IO_GAS_CABINET.DO_07_LineHeatersMC:=  GVL_COMMAND_FROM_UI.CMD_LINE_HEATER_MC_ON;

////GVL_IO_REACTOR_CABINET.DO_05_SusceptorRotationFWD:=GVL_COMMAND_FROM_UI.CMD_ROTATION_START;

//rRotationAlarm_Reset(CLK:=GVL_COMMAND_FROM_UI.CMD_ROTATION_RESET);
//IF rRotationAlarm_Reset.Q THEN
//	GVL_IO_REACTOR_CABINET.DO_05_SusceptorRotationAL_RST:=TRUE;
//END_IF

//GVL.RotationResetTon(IN:=GVL_IO_REACTOR_CABINET.DO_05_SusceptorRotationAL_RST,PT:=T#3S);

//IF GVL_IO_REACTOR_CABINET.DI_02_SusceptorRotationMotorFault = TRUE OR GVL.RotationResetTon.Q THEN
//	GVL.RotationResetTon(in:=FALSE);
//	IF GVL_IO_REACTOR_CABINET.DO_05_SusceptorRotationAL_RST = TRUE THEN
//		GVL_IO_REACTOR_CABINET.DO_05_SusceptorRotationAL_RST:=FALSE;
//	END_IF
	
//	IF GVL_IO.aOutputCmd[1].10 = TRUE THEN
//		GVL_IO.aOutputCmd[1].10:=FALSE;
//	END_IF
//END_IF


//	//GVL_IO_REACTOR_CABINET.DO_05_SusceptorRotationAL_RST:=GVL_COMMAND_FROM_UI.CMD_ROTATION_RESET;	
//GVL_IO_REACTOR_CABINET.DO_05_VacuumPumpStart_Stop := GVL_COMMAND_FROM_UI.CMD_VACUUM_PUMP_ON;
//GVL_IO_REACTOR_CABINET.DO_05_VacuumPumpReset:=GVL_COMMAND_FROM_UI.CMD_VACUUM_PUMP_RESET;

END_FUNCTION

// ---- POUs/VARIABLE_LINK/F_Variable_FromUI_Interlock.TcPOU
FUNCTION F_Variable_FromUI_Interlock: BOOL

//F_Variable_DeviceLink

END_FUNCTION

// ---- POUs/VARIABLE_LINK/F_Variable_ToUI_InputState.TcPOU
FUNCTION F_Variable_ToUI_InputState: BOOL

VAR
END_VAR

//(* UI Right Dashboard Variable*)
//GVL_IO.aInputState[1].0 := GVL_IO_REACTOR_CABINET.DI_01_MaintenanceModeKey; //Maintenance Key
//GVL_IO.aInputState[1].1	:= GVL_IO_REACTOR_CABINET.DO_06_ReactorCabinetLamp; //Reactor Cabinet Lamp
//GVL_IO.aInputState[1].2	:= GVL_IO_GAS_CABINET.DO_07_GasCabinetLamp; // Gas Cabinet Lamp
//GVL_IO.aInputState[1].3	:= GVL_IO_GAS_CABINET.DI_01_PneumaticPressureSensor; // Power Cabinet Lamp
//GVL_IO.aInputState[1].4 := GVL_IO_REACTOR_CABINET.DI_02_C_WFlowSensor; //CDA Alarm Switch
//GVL_IO.aInputState[1].5	:=GVL_IO_REACTOR_CABINET.DO_05_SusceptorRotationFWD;

//GVL_IO.aInputState[1].6 :=GVL_IO_REACTOR_CABINET.DO_05_SusceptorRotationSTOP; 
//GVL_IO.aInputState[1].7 :=NOT GVL_IO_REACTOR_CABINET.DI_02_SusceptorRotationMotorFault; //Susceptor Rotation Motor
//GVL_IO.aInputState[1].8 := GVL_IO_REACTOR_CABINET.DI_02_VacuumPumpFail; //Vacuum Pump
//GVL_IO.aInputState[1].9 := GVL_IO_REACTOR_CABINET.DI_02_VacuumPumpWarning; //Vacuum Pump
//GVL_IO.aInputState[1].10 := GVL_IO_REACTOR_CABINET.DI_02_VacuumPumpAlarm; //Vacuum Pump
//GVL_IO.aInputState[1].11 := GVL_IO_REACTOR_CABINET.DI_02_VacuumPumpFBRunning; //Vacuum Pump
//GVL_IO.aInputState[1].12 := GVL_IO_REACTOR_CABINET.DI_02_VacuumPumpFBRunning; //Vacuum Pump

//GVL_IO.aInputState[1].13 := GVL_IO_REACTOR_CABINET.DI_03_ReactorCabinetDoorClose;
//GVL_IO.aInputState[1].14 := GVL_IO_GAS_CABINET.DI_01_GasCabinetDoorClose;
//GVL_IO.aInputState[1].15 := GVL_IO_GAS_CABINET.DI_01_ControlCabinetDoorClose;

//GVL_IO.aInputState[2].0	:= GVL_IO_GAS_CABINET.DI_01_ResetButton;
//GVL_IO.aInputState[2].1	:= GVL_IO_REACTOR_CABINET.DI_02_ReactorDoorUpLimitSensor;
//GVL_IO.aInputState[2].2	:= GVL_IO_REACTOR_CABINET.DI_03_ReactorDoorDownLimitSensor;
//GVL_IO.aInputState[2].3	:= GVL_IO_REACTOR_CABINET.DI_03_CylinderAutoSwitch_Closed;
//GVL_IO.aInputState[2].4	:= GVL_IO_REACTOR_CABINET.DI_03_CylinderAutoSwitch_Opened;
//GVL_IO.aInputState[2].5	:= NOT GVL_IO_GAS_CABINET.DI_01_SMPS_1Alarm;
//GVL_IO.aInputState[2].6	:= NOT GVL_IO_GAS_CABINET.DI_01_SMPS_2Alarm;
//GVL_IO.aInputState[2].7	:= NOT GVL_IO_GAS_CABINET.DI_01_SMPS_3Alarm;
//GVL_IO.aInputState[2].8	:= NOT GVL_IO_GAS_CABINET.DI_02_SMPS_4Alarm;
//GVL_IO.aInputState[2].9	:= GVL_IO_GAS_CABINET.DI_02_GraphiteHeaterELCB;
//GVL_IO.aInputState[2].10:= GVL_IO_GAS_CABINET.DI_02_ThermalBathsELCB;
//GVL_IO.aInputState[2].11:= GVL_IO_GAS_CABINET.DI_02_VacuumPumpELCB;
//GVL_IO.aInputState[2].12:= GVL_IO_GAS_CABINET.DI_02_LineHeatersELCB;
//GVL_IO.aInputState[2].13:= GVL_IO_GAS_CABINET.DI_02_RotationMotorCP;
//GVL_IO.aInputState[2].14:= GVL_IO_GAS_CABINET.DI_02_CoverLiftMotorCP;
//GVL_IO.aInputState[2].15:= GVL_IO_GAS_CABINET.DI_02_T_VCP;

//GVL_IO.aInputState[3].0:= GVL_IO_GAS_CABINET.DI_03_GasDetectorCP;
//GVL_IO.aInputState[3].1:= GVL_IO_GAS_CABINET.DI_03_CabinetLampsCP;
//GVL_IO.aInputState[3].2:= GVL_IO_GAS_CABINET.DI_03_MFCPowerCP;
//GVL_IO.aInputState[3].3:= GVL_IO_GAS_CABINET.DI_03_LineHeater_1CP;
//GVL_IO.aInputState[3].4:= GVL_IO_GAS_CABINET.DI_03_LineHeater_2CP;
//GVL_IO.aInputState[3].5:= GVL_IO_GAS_CABINET.DI_03_LineHeater_3CP;
//GVL_IO.aInputState[3].6:= GVL_IO_GAS_CABINET.DI_03_LineHeater_4CP;
//GVL_IO.aInputState[3].7:= GVL_IO_GAS_CABINET.DI_03_LineHeater_5CP;
//GVL_IO.aInputState[3].8:= GVL_IO_GAS_CABINET.DI_04_LineHeater_6CP;
//GVL_IO.aInputState[3].9:= GVL_IO_GAS_CABINET.DI_04_LineHeater_7CP;
//GVL_IO.aInputState[3].10:= GVL_IO_GAS_CABINET.DI_04_LineHeater_8CP;

//GVL_IO.aInputState[3].11:= GVL_IO_GAS_CABINET.DI_04_GasDetectorH2;
//GVL_IO.aInputState[3].12:= GVL_IO_GAS_CABINET.DI_04_GasDetectorH2S;
//GVL_IO.aInputState[3].13:= GVL_IO_GAS_CABINET.DI_04_GasDetectorH2Se;
//GVL_IO.aInputState[3].14:= GVL_IO_GAS_CABINET.DI_04_FireSensor;
//GVL_IO.aInputState[3].15 := GVL_IO_GAS_CABINET.DI_04_ExternalScrubberFault;

//GVL_IO.aInputState[4].0 := GVL_IO_GAS_CABINET.DI_05_ExternalH2GasCabinetFault;
//GVL_IO.aInputState[4].1 := GVL_IO_GAS_CABINET.DI_05_ExternalH2SGasCabinetFault;
//GVL_IO.aInputState[4].2 := GVL_IO_GAS_CABINET.DI_05_ExternalH2SeGasCabinetFault;
//GVL_IO.aInputState[4].3 := GVL_IO_GAS_CABINET.DI_05_ExternalUserInputAlarm;

//GVL_IO.aInputState[4].4:= GVL_IO_GAS_CABINET.DI_05_ThermalBath_1DeviationAlarm;
//GVL_IO.aInputState[4].5:= GVL_IO_GAS_CABINET.DI_05_ThermalBath_1CutOffAlarm;
//GVL_IO.aInputState[4].6:= GVL_IO_GAS_CABINET.DI_05_ThermalBath_2DeviationAlarm;
//GVL_IO.aInputState[4].7:= GVL_IO_GAS_CABINET.DI_05_ThermalBath_2CutOffAlarm;
//GVL_IO.aInputState[4].8:= GVL_IO_GAS_CABINET.DI_06_ThermalBath_3DeviationAlarm;
//GVL_IO.aInputState[4].9:= GVL_IO_GAS_CABINET.DI_06_ThermalBath_3CutOffAlarm;
//GVL_IO.aInputState[4].10:= GVL_IO_GAS_CABINET.DI_06_ThermalBath_4DeviationAlarm;
//GVL_IO.aInputState[4].11:= GVL_IO_GAS_CABINET.DI_06_ThermalBath_3CutOffAlarm;


//GVL_IO.aInputState[5].0:= GVL_IO_REACTOR_CABINET.DO_04_SignalTowerRed;
//GVL_IO.aInputState[5].1:= GVL_IO_REACTOR_CABINET.DO_04_SignalTowerOrange;
//GVL_IO.aInputState[5].2:= GVL_IO_REACTOR_CABINET.DO_04_SignalTowerGreen;
//GVL_IO.aInputState[5].3:= GVL_IO_REACTOR_CABINET.DO_04_SignalTowerBlue;
//GVL_IO.aInputState[5].4:= GVL_IO_REACTOR_CABINET.DO_04_SignalTowerWhite;
//GVL_IO.aInputState[5].5:= GVL_IO_REACTOR_CABINET.DO_04_SignalTowerBuzzer;

//GVL_IO.aInputState[5].6:= GVL_IO_REACTOR_CABINET.DI_01_ClampLock;
//GVL_IO.aInputState[5].7:= GVL_IO_REACTOR_CABINET.DI_01_ClampRelease;

//GVL_IO.aInputState[5].8:= F_GetDorPressure(GVL_IO_REACTOR_CABINET.AI_07_S05_DORPressurePV) < 100;
//GVL_IO.aInputState[5].9:= GVL_DEVICE_NET_E3508.aInputAlarmStatus[1] > 0 OR GVL_DEVICE_NET_E3508.aInputAlarmStatus[2] > 0 ;
//GVL_IO.aInputState[5].10:= GVL_DEVICE_NET_E3508.aInputManAutoBytes[1].0;//(*True:manual   False:auto*)

//GVL_IO.aInputState[6].0:= GVL_DEVICE_NET_IQ_PLUS.nInputStatus  = 0;
//GVL_IO.aInputState[6].1:= GVL_DEVICE_NET_IQ_PLUS.nInputStatus  = 1;
//GVL_IO.aInputState[6].2:= GVL_DEVICE_NET_IQ_PLUS.nInputStatus  = 2;
//GVL_IO.aInputState[6].3:= GVL_DEVICE_NET_IQ_PLUS.nInputStatus  = 3;
//GVL_IO.aInputState[6].4:= GVL_DEVICE_NET_IQ_PLUS.nInputStatus  = 4;
//GVL_IO.aInputState[6].5:= GVL_DEVICE_NET_IQ_PLUS.nInputStatus  = 5;
//GVL_IO.aInputState[6].6:= GVL_DEVICE_NET_IQ_PLUS.nInputStatus  = 6;
//GVL_IO.aInputState[6].7:= GVL_DEVICE_NET_IQ_PLUS.nInputStatus  = 7;
//GVL_IO.aInputState[6].8:= GVL_DEVICE_NET_IQ_PLUS.nInputStatus  = 8;

//GVL_IO.aInputState[6].9:= P90_Interlock.bRecipeStartAvailable;
//GVL_IO.aInputState[6].10:= P90_Interlock.bReactorOpenEnable;
//GVL_IO.aInputState[6].12:= GVL_IO_REACTOR_CABINET.DI_03_ReactorDoorDownLimitSensor AND P90_Interlock.AlarmTrig = FALSE AND GVL_IO_VALVE.DO_00_V21PumpByPass = FALSE;

END_FUNCTION

// ---- POUs/P11_E3508.TcPOU
PROGRAM P11_E3508
VAR
	wControlValue			: WORD;
	wPowerRateSetValue		: WORD;	
	bOutputManAuto 			: BOOL; // Command 0:Auto, 1:Manual Mode
	
	bHeaterOn				: BOOL := FALSE; //to PSTEK
	bHeaterReset			: BOOL; //to PSTEK

	bAlarmState_E3508 		: BOOL; //Alarm or Sensor Break Signal
	bManAuto_E3508 			: BOOL; //State, 0:Manual, 1:Auto

	isHeaterReady			: BOOL; //Close : Ready
	isHeaterRun				: BOOL; //Close : Running, Open : Stop
	isHeaterFault			: BOOL; //Close : Falut, Open : Normal
	//isInductionHeaterErr	: BOOL; //Power Supply
	bInductionHeaterCB		: BOOL;
	//Input from E3508 Controller
//	aInputPVBytes AT %I* 		: ARRAY[1..2]OF USINT; //Input Process Values
//	aInputSVBytes AT %I* 		: ARRAY[1..2]OF USINT; //Input Set Values
//	aInputTVBytes AT %I* 		: ARRAY[1..2]OF USINT; //Input Target Valuse
//	aInputCVBytes AT %I* 		: ARRAY[1..2]OF USINT; //Induction Heter Controlled Values
//	aInputProportional AT %I* 	: ARRAY[1..2]OF USINT; //PID - Proportional Band
//	aInputIntegral AT %I* 		: ARRAY[1..2]OF USINT; //PID - Integral Time
//	aInputDerivative AT %I* 	: ARRAY[1..2]OF USINT; //PID - Derivative Time 
//	nInputAlarmBytes AT %I* 	: USINT; // Alarm State
//	nInputManAutoBytes AT %I* 	: USINT; // ManAuto State
	
	wE3508_PV				: WORD;
	wE3508_SV				: WORD;
	wE3508_PowerRate		: WORD; //To Induction Heater Control Values
	wE3508_P				: WORD; //PID Parameter P
	wE3508_I				: WORD; //PID Parameter I
	wE3508_D				: WORD; //PID Parameter D
	//Output to E3508 Controller
	wOutputSVBytes 				: outWord;
	wOutputPowerSVBytes 		: outWord;

END_VAR

//jhkang_251112
////Induction Heater & Temperature Controller & Thermo Couple(R-Type)
////Maker: PSTEK, Eurotherm
////Model: 3508
////Temperature Range: 0 ~ 12000℃

//(* Command *)
//bHeaterOn := GVL_COMMAND_FROM_UI.CMD_HEATER_MAIN_MC_ON;


//GVL_DEVICE_NET_E3508.nOutputManAutoBytes[1].0 := GVL_COMMAND_FROM_UI.CMD_E3508_MAN_AUTO; //Temp Controller Mode Command(*True:manual   False:auto*)

//(* Read from Power Distribution Pannel *)
//bInductionHeaterCB		:= GVL_IO_GAS_CABINET.DI_02_GraphiteHeaterELCB;

//(* Read from E3508 Device Value *)
//wE3508_PV				:= USINT_TO_WORD_Bit(GVL_DEVICE_NET_E3508.aInputPVBytes[1], GVL_DEVICE_NET_E3508.aInputPVBytes[2]);
//wE3508_SV				:= USINT_TO_WORD_Bit(GVL_DEVICE_NET_E3508.aInputSVBytes[1], GVL_DEVICE_NET_E3508.aInputSVBytes[2]);
//wE3508_PowerRate		:= USINT_TO_WORD_Bit(GVL_DEVICE_NET_E3508.aInputActiveOut[1], GVL_DEVICE_NET_E3508.aInputActiveOut[2]); //divided to 10

//wE3508_P 				:= USINT_TO_WORD_Bit(GVL_DEVICE_NET_E3508.aInputProportional[1], GVL_DEVICE_NET_E3508.aInputProportional[2]);
//wE3508_I 				:= USINT_TO_WORD_Bit(GVL_DEVICE_NET_E3508.aInputIntegral[1], GVL_DEVICE_NET_E3508.aInputIntegral[2]);
//wE3508_D 				:= USINT_TO_WORD_Bit(GVL_DEVICE_NET_E3508.aInputDerivative[1], GVL_DEVICE_NET_E3508.aInputDerivative[2]);



////bAlarmState_E3508 		:= nInputAlarmBytes.7;

////GVL_INTERFACE_UI.aMonitoring_PV[11] := WORD_TO_REAL(wE3508_PowerRate)*0.1; //divided to 10 PowerRate

//(* Read from Induction Heater Value *)

//// Interface with other PRGs
//wControlValue			:= GVL_IO.wE3508_CV;
//GVL_IO.wE3508_PV		:= wE3508_PV;

//(* Write to E3508 Device Value *)
//// Operation Mode
//// bOutputManAuto := GVL_IO.aOutputCmd[1].11; //Temp Controller Mode Command
//// nOutputManAutoBytes.0 	:= GVL_IO.aOutputCmd[1].11; //Command

//IF GVL_DEVICE_NET_E3508.aInputManAutoBytes[1].0 THEN // Read form E3508 Mode, 0:Man 1:Auto
//	wOutputPowerSVBytes 	:= WORD_TO_USINT_Bit(wControlValue); //multiple to 10, Power Reate Set Value
//	GVL_DEVICE_NET_E3508.aOutputPowerBytes[1] 	:= wOutputPowerSVBytes.Lower;
//	GVL_DEVICE_NET_E3508.aOutputPowerBytes[2] 	:= wOutputPowerSVBytes.Upper;
//ELSE
//	wOutputSVBytes 			:= WORD_TO_USINT_Bit(wControlValue / 10 ); // Temperature Set Value
//	GVL_DEVICE_NET_E3508.aOutputSVBytes[1] 		:= wOutputSVBytes.Lower;
//	GVL_DEVICE_NET_E3508.aOutputSVBytes[2] 		:= wOutputSVBytes.Upper;
//END_IF

//(* Write to Induction Heater Value *)
//GVL_IO_GAS_CABINET.DO_07_GraphiteHeaterMC := bHeaterOn;
////GVL_IO.aDigitalOutputIO[2].1 := bHeaterReset;
//GVL_IO.nE3508_nInputManAutoBytes := GVL_DEVICE_NET_E3508.aInputManAutoBytes[1]; //State


//GVL_DEVICE_NET_E3508.aOutputThreshold[1]:=232;
//GVL_DEVICE_NET_E3508.aOutputThreshold[2]:=3;

END_PROGRAM

// ---- POUs/P12_IQ_PLUS.TcPOU
PROGRAM P12_IQ_PLUS
VAR
	wControlValue 		: WORD := 760;//Pressure Set Value
	wCDG1_PV 			: WORD; //CD2 Current Pressure
	wCDG2_PV 			: WORD; //CD2 Current Pressure
	bVacuumPumpCB		: BOOL;
	bThrottleValveCP	: BOOL;

